(* Logix 5000 project; controller CarbonScout_MK6 vendor 1 type 14 code 154 rev 32.11; software revision 32.00; part 7 of 17 *)

        [2,16].Day := 20, [2,16].Month := 11, [2,16].Year := 2021, [2,16].Sample_DO := 5.8144927, [2,16].Sample_pH := 9.2394, [2,16].Sample_VOL := 17.577055, [2,16].Density := 412.98294, [2,16].EmptyDist := 1410.0, [2,16].FullDist := 1326.2568, [2,16].Carbon_mLperL := 12.587779, [2,16].Slurry_Weight := -10.52187, [2,16].Sample_Tank := 2, [2,16].Carbon_Height := 83.743164, [2,16].Sample_FlowRate := 1.5023123, [2,16].Sample_FillTime := 11.700001, [2,16].DisplacedCarbonVol := 1512.862, [2,16].DisplacedCarbonMass := 756.431, [2,16].SampleDuration := 964, [2,17].Run_ID := 2610, [2,17].Carbon_VOL_ml := 220.35596, [2,17].Carbon_MASS := 110.17798, [2,17].Carbon_DIST := 6.5356975, [2,17].Hour := 1, [2,17].Min := 21, [2,17].Day := 20, [2,17].Month := 11, [2,17].Year := 2021, [2,17].Sample_DO := 6.0987396, [2,17].Sample_pH := 9.333745, [2,17].Sample_VOL := 16.857876, [2,17].Density := 402.41284, [2,17].EmptyDist := 1410.0, [2,17].FullDist := 1326.5975, [2,17].Carbon_mLperL := 13.071395, [2,17].Slurry_Weight := -10.52187, [2,17].Sample_Tank := 2, [2,17].Carbon_Height := 83.402466, [2,17].Sample_FlowRate := 1.9698381, [2,17].Sample_FillTime := 8.558001, [2,17].DisplacedCarbonVol := 2059.8826, [2,17].DisplacedCarbonMass := 1029.9413, [2,17].SampleDuration := 1054, [2,18].Run_ID := 2601, [2,18].Carbon_VOL_ml := 180.58542, [2,18].Carbon_MASS := 90.29271, [2,18].Carbon_DIST := 5.3398423, [2,18].Hour := 23, [2,18].Min := 4, [2,18].Day := 19, [2,18].Month := 11, [2,18].Year := 2021, [2,18].Sample_DO := 6.4815454, [2,18].Sample_pH := 9.355976, [2,18].Sample_VOL := 16.909246, [2,18].Density := 403.16788, [2,18].EmptyDist := 1410.0, [2,18].FullDist := 1341.6503, [2,18].Carbon_mLperL := 10.679685, [2,18].Slurry_Weight := -10.52187, [2,18].Sample_Tank := 2,
        [2,18].Carbon_Height := 68.34973, [2,18].Sample_FlowRate := 2.087561, [2,18].Sample_FillTime := 8.100001, [2,18].DisplacedCarbonVol := 1783.5593, [2,18].DisplacedCarbonMass := 891.77966, [2,18].SampleDuration := 876, [2,19].Run_ID := 2593, [2,19].Carbon_VOL_ml := 185.95343, [2,19].Carbon_MASS := 92.976715, [2,19].Carbon_DIST := 5.4190025, [2,19].Hour := 21, [2,19].Min := 7, [2,19].Day := 19, [2,19].Month := 11, [2,19].Year := 2021, [2,19].Sample_DO := 6.719078, [2,19].Sample_pH := 9.30912, [2,19].Sample_VOL := 17.157534, [2,19].Density := 406.81705, [2,19].EmptyDist := 1410.0, [2,19].FullDist := 1339.6185, [2,19].Carbon_mLperL := 10.838005, [2,19].Slurry_Weight := -10.52187, [2,19].Sample_Tank := 2, [2,19].Carbon_Height := 70.38147, [2,19].Sample_FlowRate := 2.3369017, [2,19].Sample_FillTime := 7.342001, [2,19].DisplacedCarbonVol := 2026.1881, [2,19].DisplacedCarbonMass := 1013.09406, [2,19].SampleDuration := 876, [3,0].Run_ID := 2785, [3,0].Hour := 22, [3,0].Min := 56, [3,0].Day := 21, [3,0].Month := 11, [3,0].Year := 2021, [3,0].Sample_DO := 5.975054, [3,0].Sample_pH := 9.085041, [3,0].Sample_VOL := 17.71404, [3,0].Density := 414.99634, [3,0].EmptyDist := 1410.0, [3,0].FullDist := 1441.737, [3,0].ErrorFlag := 1, [3,0].Slurry_Weight := -10.52187, [3,0].Sample_Tank := 3, [3,0].Carbon_Height := -31.73706, [3,0].Sample_FlowRate := 1.3902087, [3,0].Sample_FillTime := 12.742001, [3,0].SampleDuration := 926, [3,1].Run_ID := 2784, [3,1].Carbon_VOL_ml := 131.5602, [3,1].Carbon_MASS := 65.7801, [3,1].Carbon_DIST := 3.8647463, [3,1].Hour := 22, [3,1].Min := 41, [3,1].Day := 21, [3,1].Month := 11, [3,1].Year := 2021, [3,1].Sample_DO := 6.334731, [3,1].Sample_pH := 9.09235,
        [3,1].Sample_VOL := 17.020548, [3,1].Density := 404.8037, [3,1].EmptyDist := 1410.0, [3,1].FullDist := 1360.2058, [3,1].Carbon_mLperL := 7.7294927, [3,1].Slurry_Weight := -10.52187, [3,1].Sample_Tank := 3, [3,1].Carbon_Height := 49.79419, [3,1].Sample_FlowRate := 1.350837, [3,1].Sample_FillTime := 12.600001, [3,1].DisplacedCarbonVol := 1044.1285, [3,1].DisplacedCarbonMass := 522.0643, [3,1].SampleDuration := 941, [3,2].Run_ID := 2771, [3,2].Hour := 19, [3,2].Min := 27, [3,2].Day := 21, [3,2].Month := 11, [3,2].Year := 2021, [3,2].Sample_DO := 6.247068, [3,2].Sample_pH := 9.097762, [3,2].Sample_VOL := 17.619864, [3,2].Density := 413.61212, [3,2].EmptyDist := 1410.0, [3,2].FullDist := 1446.4924, [3,2].ErrorFlag := 1, [3,2].Slurry_Weight := -10.52187, [3,2].Sample_Tank := 3, [3,2].Carbon_Height := -36.49243, [3,2].Sample_FlowRate := 1.4161599, [3,2].Sample_FillTime := 12.442001, [3,2].SampleDuration := 925, [3,3].Run_ID := 2770, [3,3].Hour := 19, [3,3].Min := 12, [3,3].Day := 21, [3,3].Month := 11, [3,3].Year := 2021, [3,3].Sample_DO := 5.9098787, [3,3].Sample_pH := 9.116793, [3,3].Sample_VOL := 16.515411, [3,3].Density := 397.3795, [3,3].EmptyDist := 1410.0, [3,3].FullDist := 1444.21, [3,3].Slurry_Weight := -10.52187, [3,3].Sample_Tank := 3, [3,3].Carbon_Height := -34.20996, [3,3].Sample_FlowRate := 1.428916, [3,3].Sample_FillTime := 11.558001, [3,3].SampleDuration := 988, [3,4].Run_ID := 2748, [3,4].Carbon_VOL_ml := 107.38028, [3,4].Carbon_MASS := 53.69014, [3,4].Carbon_DIST := 3.1075363, [3,4].Hour := 13, [3,4].Min := 17, [3,4].Day := 21, [3,4].Month := 11, [3,4].Year := 2021, [3,4].Sample_DO := 6.1838565,
        [3,4].Sample_pH := 9.131414, [3,4].Sample_VOL := 17.277397, [3,4].Density := 408.57877, [3,4].EmptyDist := 1410.0, [3,4].FullDist := 1369.3577, [3,4].ErrorFlag := 1, [3,4].Carbon_mLperL := 6.2150726, [3,4].Slurry_Weight := -10.52187, [3,4].Sample_Tank := 3, [3,4].Carbon_Height := 40.642334, [3,4].Sample_FlowRate := 1.1410247, [3,4].Sample_FillTime := 15.142001, [3,4].DisplacedCarbonVol := 709.15515, [3,4].DisplacedCarbonMass := 354.57758, [3,4].SampleDuration := 928, [3,5].Run_ID := 2747, [3,5].Carbon_VOL_ml := 89.66557, [3,5].Carbon_MASS := 44.832787, [3,5].Carbon_DIST := 2.55687, [3,5].Hour := 13, [3,5].Min := 1, [3,5].Day := 21, [3,5].Month := 11, [3,5].Year := 2021, [3,5].Sample_DO := 5.9852405, [3,5].Sample_pH := 9.164311, [3,5].Sample_VOL := 17.534246, [3,5].Density := 412.35376, [3,5].EmptyDist := 1410.0, [3,5].FullDist := 1376.0625, [3,5].Carbon_mLperL := 5.11374, [3,5].Slurry_Weight := -10.52187, [3,5].Sample_Tank := 3, [3,5].Carbon_Height := 33.9375, [3,5].Sample_FlowRate := 1.1354905, [3,5].Sample_FillTime := 15.442001, [3,5].DisplacedCarbonVol := 580.66034, [3,5].DisplacedCarbonMass := 290.33017, [3,5].SampleDuration := 876, [3,6].Run_ID := 2734, [3,6].Carbon_VOL_ml := 232.73778, [3,6].Carbon_MASS := 116.36889, [3,6].Carbon_DIST := 6.594802, [3,6].Hour := 9, [3,6].Min := 47, [3,6].Day := 21, [3,6].Month := 11, [3,6].Year := 2021, [3,6].Sample_DO := 5.8418803, [3,6].Sample_pH := 9.115876, [3,6].Sample_VOL := 17.645548, [3,6].Density := 413.98962, [3,6].EmptyDist := 1410.0, [3,6].FullDist := 1321.9111, [3,6].ErrorFlag := 1, [3,6].Carbon_mLperL := 13.189604, [3,6].Slurry_Weight := -10.52187, [3,6].Sample_Tank := 3, [3,6].Carbon_Height := 88.08887, [3,6].Sample_FlowRate := 1.2389796,
        [3,6].Sample_FillTime := 14.242001, [3,6].DisplacedCarbonVol := 1634.165, [3,6].DisplacedCarbonMass := 817.0825, [3,6].SampleDuration := 927, [3,7].Run_ID := 2733, [3,7].Carbon_VOL_ml := 232.98547, [3,7].Carbon_MASS := 116.49274, [3,7].Carbon_DIST := 6.776072, [3,7].Hour := 9, [3,7].Min := 31, [3,7].Day := 21, [3,7].Month := 11, [3,7].Year := 2021, [3,7].Sample_DO := 6.0491557, [3,7].Sample_pH := 9.1932335, [3,7].Sample_VOL := 17.19178, [3,7].Density := 407.3204, [3,7].EmptyDist := 1410.0, [3,7].FullDist := 1321.8174, [3,7].Carbon_mLperL := 13.552144, [3,7].Slurry_Weight := -10.52187, [3,7].Sample_Tank := 3, [3,7].Carbon_Height := 88.18262, [3,7].Sample_FlowRate := 1.3326961, [3,7].Sample_FillTime := 12.900001, [3,7].DisplacedCarbonVol := 1806.0889, [3,7].DisplacedCarbonMass := 903.04443, [3,7].SampleDuration := 877, [3,8].Run_ID := 2723, [3,8].Carbon_VOL_ml := 140.70815, [3,8].Carbon_MASS := 70.35407, [3,8].Carbon_DIST := 3.9870722, [3,8].Hour := 6, [3,8].Min := 9, [3,8].Day := 21, [3,8].Month := 11, [3,8].Year := 2021, [3,8].Sample_DO := 5.5555353, [3,8].Sample_pH := 9.267746, [3,8].Sample_VOL := 17.645548, [3,8].Density := 413.98962, [3,8].EmptyDist := 1410.0, [3,8].FullDist := 1356.7434, [3,8].Carbon_mLperL := 7.9741445, [3,8].Slurry_Weight := -10.52187, [3,8].Sample_Tank := 3, [3,8].Carbon_Height := 53.25659, [3,8].Sample_FlowRate := 1.5896888, [3,8].Sample_FillTime := 11.100001, [3,8].DisplacedCarbonVol := 1267.6407, [3,8].DisplacedCarbonMass := 633.8204, [3,8].SampleDuration := 872, [3,9].Run_ID := 2712, [3,9].Carbon_VOL_ml := 180.66768, [3,9].Carbon_MASS := 90.33384, [3,9].Carbon_DIST := 5.0995617, [3,9].Hour := 3, [3,9].Min := 23, [3,9].Day := 21, [3,9].Month := 11,
        [3,9].Year := 2021, [3,9].Sample_DO := 6.18531, [3,9].Sample_pH := 9.155949, [3,9].Sample_VOL := 17.71404, [3,9].Density := 414.99634, [3,9].EmptyDist := 1410.0, [3,9].FullDist := 1341.6191, [3,9].Carbon_mLperL := 10.199123, [3,9].Slurry_Weight := -10.52187, [3,9].Sample_Tank := 3, [3,9].Carbon_Height := 68.38086, [3,9].Sample_FlowRate := 1.4958655, [3,9].Sample_FillTime := 11.842001, [3,9].DisplacedCarbonVol := 1525.6516, [3,9].DisplacedCarbonMass := 762.8258, [3,9].SampleDuration := 874, [3,10].Run_ID := 2701, [3,10].Carbon_VOL_ml := 169.69102, [3,10].Carbon_MASS := 84.84551, [3,10].Carbon_DIST := 4.8721514, [3,10].Min := 44, [3,10].Day := 21, [3,10].Month := 11, [3,10].Year := 2021, [3,10].Sample_DO := 5.931424, [3,10].Sample_pH := 9.080997, [3,10].Sample_VOL := 17.414383, [3,10].Density := 410.59213, [3,10].EmptyDist := 1410.0, [3,10].FullDist := 1345.7737, [3,10].ErrorFlag := 1, [3,10].Carbon_mLperL := 9.744303, [3,10].Slurry_Weight := -10.52187, [3,10].Sample_Tank := 3, [3,10].Carbon_Height := 64.22632, [3,10].Sample_FlowRate := 1.3666915, [3,10].Sample_FillTime := 12.742001, [3,10].DisplacedCarbonVol := 1331.7456, [3,10].DisplacedCarbonMass := 665.8728, [3,10].SampleDuration := 927, [3,11].Run_ID := 2700, [3,11].Carbon_VOL_ml := 162.94458, [3,11].Carbon_MASS := 81.47229, [3,11].Carbon_DIST := 4.5357313, [3,11].Min := 28, [3,11].Day := 21, [3,11].Month := 11, [3,11].Year := 2021, [3,11].Sample_DO := 6.049618, [3,11].Sample_pH := 9.090882, [3,11].Sample_VOL := 17.962328, [3,11].Density := 418.64548, [3,11].EmptyDist := 1410.0, [3,11].FullDist := 1348.3271, [3,11].Carbon_mLperL := 9.071463, [3,11].Slurry_Weight := -10.52187, [3,11].Sample_Tank := 3, [3,11].Carbon_Height := 61.67285, [3,11].Sample_FlowRate := 1.3305427, [3,11].Sample_FillTime := 13.500001,
        [3,11].DisplacedCarbonVol := 1206.997, [3,11].DisplacedCarbonMass := 603.4985, [3,11].SampleDuration := 877, [3,12].Run_ID := 2688, [3,12].Carbon_VOL_ml := 2.5427434, [3,12].Carbon_MASS := 1.2713717, [3,12].Carbon_DIST := 0.071323834, [3,12].Hour := 21, [3,12].Min := 31, [3,12].Day := 20, [3,12].Month := 11, [3,12].Year := 2021, [3,12].Sample_DO := 5.966387, [3,12].Sample_pH := 9.127291, [3,12].Sample_VOL := 17.825342, [3,12].Density := 416.63214, [3,12].EmptyDist := 1410.0, [3,12].FullDist := 1409.0376, [3,12].ErrorFlag := 1, [3,12].Carbon_mLperL := 0.14264767, [3,12].Slurry_Weight := -10.52187, [3,12].Sample_Tank := 3, [3,12].Carbon_Height := 0.96240234, [3,12].Sample_FlowRate := 1.5052644, [3,12].Sample_FillTime := 11.842001, [3,12].DisplacedCarbonVol := 21.472246, [3,12].DisplacedCarbonMass := 10.736123, [3,12].SampleDuration := 926, [3,13].Run_ID := 2687, [3,13].Carbon_VOL_ml := 87.715294, [3,13].Carbon_MASS := 43.857647, [3,13].Carbon_DIST := 2.512297, [3,13].Hour := 21, [3,13].Min := 16, [3,13].Day := 20, [3,13].Month := 11, [3,13].Year := 2021, [3,13].Sample_DO := 6.0653386, [3,13].Sample_pH := 9.228728, [3,13].Sample_VOL := 17.457191, [3,13].Density := 411.22125, [3,13].EmptyDist := 1410.0, [3,13].FullDist := 1376.8007, [3,13].Carbon_mLperL := 5.024594, [3,13].Slurry_Weight := -10.52187, [3,13].Sample_Tank := 3, [3,13].Carbon_Height := 33.19934, [3,13].Sample_FlowRate := 1.4741758, [3,13].Sample_FillTime := 11.842001, [3,13].DisplacedCarbonVol := 740.7135, [3,13].DisplacedCarbonMass := 370.35675, [3,13].SampleDuration := 873, [3,14].Run_ID := 2676, [3,14].Carbon_VOL_ml := 316.40967, [3,14].Carbon_MASS := 158.20483, [3,14].Carbon_DIST := 9.120595, [3,14].Hour := 18, [3,14].Min := 27, [3,14].Day := 20, [3,14].Month := 11,
        [3,14].Year := 2021, [3,14].Sample_DO := 5.684902, [3,14].Sample_pH := 9.152988, [3,14].Sample_VOL := 17.34589, [3,14].Density := 409.58542, [3,14].EmptyDist := 1410.0, [3,14].FullDist := 1290.2422, [3,14].ErrorFlag := 1, [3,14].Carbon_mLperL := 18.24119, [3,14].Slurry_Weight := -10.52187, [3,14].Sample_Tank := 3, [3,14].Carbon_Height := 119.75781, [3,14].Sample_FlowRate := 1.5626926, [3,14].Sample_FillTime := 11.100001, [3,14].DisplacedCarbonVol := 2850.5374, [3,14].DisplacedCarbonMass := 1425.2687, [3,14].SampleDuration := 925, [3,15].Run_ID := 2675, [3,15].Carbon_VOL_ml := 318.91373, [3,15].Carbon_MASS := 159.45686, [3,15].Carbon_DIST := 9.321602, [3,15].Hour := 18, [3,15].Min := 11, [3,15].Day := 20, [3,15].Month := 11, [3,15].Year := 2021, [3,15].Sample_DO := 5.655153, [3,15].Sample_pH := 9.277301, [3,15].Sample_VOL := 17.106165, [3,15].Density := 406.06207, [3,15].EmptyDist := 1410.0, [3,15].FullDist := 1289.2944, [3,15].Carbon_mLperL := 18.643204, [3,15].Slurry_Weight := -10.52187, [3,15].Sample_Tank := 3, [3,15].Carbon_Height := 120.70557, [3,15].Sample_FlowRate := 1.5005407, [3,15].Sample_FillTime := 11.400001, [3,15].DisplacedCarbonVol := 2797.4888, [3,15].DisplacedCarbonMass := 1398.7444, [3,15].SampleDuration := 871, [3,16].Run_ID := 2663, [3,16].Carbon_VOL_ml := 193.90451, [3,16].Carbon_MASS := 96.952255, [3,16].Carbon_DIST := 5.6338425, [3,16].Hour := 15, [3,16].Min := 17, [3,16].Day := 20, [3,16].Month := 11, [3,16].Year := 2021, [3,16].Sample_DO := 5.4973636, [3,16].Sample_pH := 9.102047, [3,16].Sample_VOL := 17.208904, [3,16].Density := 407.57208, [3,16].EmptyDist := 1410.0, [3,16].FullDist := 1336.6091, [3,16].ErrorFlag := 1, [3,16].Carbon_mLperL := 11.267685, [3,16].Slurry_Weight := -10.52187, [3,16].Sample_Tank := 3,
        [3,16].Carbon_Height := 73.39087, [3,16].Sample_FlowRate := 1.4173038, [3,16].Sample_FillTime := 12.142001, [3,16].DisplacedCarbonVol := 1596.9734, [3,16].DisplacedCarbonMass := 798.4867, [3,16].SampleDuration := 925, [3,17].Run_ID := 2662, [3,17].Hour := 15, [3,17].Min := 1, [3,17].Day := 20, [3,17].Month := 11, [3,17].Year := 2021, [3,17].Sample_DO := 5.5800033, [3,17].Sample_pH := 9.173197, [3,17].Sample_VOL := 17.55993, [3,17].Density := 412.73126, [3,17].EmptyDist := 1410.0, [3,17].FullDist := 1430.6094, [3,17].Slurry_Weight := -10.52187, [3,17].Sample_Tank := 3, [3,17].Carbon_Height := -20.609375, [3,17].Sample_FlowRate := 1.4276365, [3,17].Sample_FillTime := 12.300001, [3,17].SampleDuration := 872, [3,18].Run_ID := 2650, [3,18].Carbon_VOL_ml := 169.7033, [3,18].Carbon_MASS := 84.85165, [3,18].Carbon_DIST := 5.056465, [3,18].Hour := 12, [3,18].Day := 20, [3,18].Month := 11, [3,18].Year := 2021, [3,18].Sample_DO := 5.6071215, [3,18].Sample_pH := 9.084224, [3,18].Sample_VOL := 16.780823, [3,18].Density := 401.2804, [3,18].EmptyDist := 1410.0, [3,18].FullDist := 1345.769, [3,18].Carbon_mLperL := 10.11293, [3,18].Slurry_Weight := -10.52187, [3,18].Sample_Tank := 3, [3,18].Carbon_Height := 64.23096, [3,18].Sample_FlowRate := 1.1187215, [3,18].Sample_FillTime := 15.000001, [3,18].DisplacedCarbonVol := 1131.3552, [3,18].DisplacedCarbonMass := 565.6776, [3,18].SampleDuration := 878, [3,19].Run_ID := 2640, [3,19].Carbon_VOL_ml := 185.8657, [3,19].Carbon_MASS := 92.93285, [3,19].Carbon_DIST := 5.354986, [3,19].Hour := 9, [3,19].Min := 28, [3,19].Day := 20, [3,19].Month := 11, [3,19].Year := 2021, [3,19].Sample_DO := 6.2630897, [3,19].Sample_pH := 9.137375, [3,19].Sample_VOL := 17.354452, [3,19].Density := 409.71127,
        [3,19].EmptyDist := 1410.0, [3,19].FullDist := 1339.6517, [3,19].Carbon_mLperL := 10.709972, [3,19].Slurry_Weight := -10.52187, [3,19].Sample_Tank := 3, [3,19].Carbon_Height := 70.34827, [3,19].Sample_FlowRate := 1.1226841, [3,19].Sample_FillTime := 15.458001, [3,19].DisplacedCarbonVol := 1202.3916, [3,19].DisplacedCarbonMass := 601.1958, [3,19].SampleDuration := 879, [4,0].Run_ID := 2787, [4,0].Hour := 23, [4,0].Min := 27, [4,0].Day := 21, [4,0].Month := 11, [4,0].Year := 2021, [4,0].Sample_DO := 5.6127687, [4,0].Sample_pH := 9.112585, [4,0].Sample_VOL := 17.34589, [4,0].Density := 409.58542, [4,0].EmptyDist := 1410.0, [4,0].FullDist := 1447.225, [4,0].ErrorFlag := 1, [4,0].Slurry_Weight := -10.52187, [4,0].Sample_Tank := 4, [4,0].Carbon_Height := -37.224976, [4,0].Sample_FlowRate := 1.464777, [4,0].Sample_FillTime := 11.842001, [4,0].SampleDuration := 926, [4,1].Run_ID := 2786, [4,1].Hour := 23, [4,1].Min := 11, [4,1].Day := 21, [4,1].Month := 11, [4,1].Year := 2021, [4,1].Sample_DO := 5.879518, [4,1].Sample_pH := 9.193804, [4,1].Sample_VOL := 17.208904, [4,1].Density := 407.57208, [4,1].EmptyDist := 1410.0, [4,1].FullDist := 1447.1635, [4,1].Slurry_Weight := -10.52187, [4,1].Sample_Tank := 4, [4,1].Carbon_Height := -37.163452, [4,1].Sample_FlowRate := 1.4340752, [4,1].Sample_FillTime := 12.000001, [4,1].SampleDuration := 927, [4,2].Run_ID := 2773, [4,2].Hour := 19, [4,2].Min := 58, [4,2].Day := 21, [4,2].Month := 11, [4,2].Year := 2021, [4,2].Sample_DO := 5.849701, [4,2].Sample_pH := 9.101484, [4,2].Sample_VOL := 17.722603, [4,2].Density := 415.12213, [4,2].EmptyDist := 1410.0, [4,2].FullDist := 1447.1489,
        [4,2].ErrorFlag := 1, [4,2].Slurry_Weight := -10.52187, [4,2].Sample_Tank := 4, [4,2].Carbon_Height := -37.148926, [4,2].Sample_FlowRate := 1.3127853, [4,2].Sample_FillTime := 13.500001, [4,2].SampleDuration := 927, [4,3].Run_ID := 2772, [4,3].Hour := 19, [4,3].Min := 43, [4,3].Day := 21, [4,3].Month := 11, [4,3].Year := 2021, [4,3].Sample_DO := 5.853695, [4,3].Sample_pH := 9.12075, [4,3].Sample_VOL := 17.465754, [4,3].Density := 411.34714, [4,3].EmptyDist := 1410.0, [4,3].FullDist := 1440.5786, [4,3].Slurry_Weight := -10.52187, [4,3].Sample_Tank := 4, [4,3].Carbon_Height := -30.578613, [4,3].Sample_FlowRate := 1.3391927, [4,3].Sample_FillTime := 13.042001, [4,3].SampleDuration := 926, [4,4].Run_ID := 2750, [4,4].Carbon_VOL_ml := 178.94606, [4,4].Carbon_MASS := 89.47303, [4,4].Carbon_DIST := 5.1940603, [4,4].Hour := 13, [4,4].Min := 48, [4,4].Day := 21, [4,4].Month := 11, [4,4].Year := 2021, [4,4].Sample_DO := 5.656315, [4,4].Sample_pH := 9.1106205, [4,4].Sample_VOL := 17.226028, [4,4].Density := 407.82376, [4,4].EmptyDist := 1410.0, [4,4].FullDist := 1342.2708, [4,4].ErrorFlag := 1, [4,4].Carbon_mLperL := 10.388121, [4,4].Slurry_Weight := -10.52187, [4,4].Sample_Tank := 4, [4,4].Carbon_Height := 67.72925, [4,4].Sample_FlowRate := 1.0350935, [4,4].Sample_FillTime := 16.642002, [4,4].DisplacedCarbonVol := 1075.2677, [4,4].DisplacedCarbonMass := 537.63385, [4,4].SampleDuration := 931, [4,5].Run_ID := 2749, [4,5].Hour := 13, [4,5].Min := 32, [4,5].Day := 21, [4,5].Month := 11, [4,5].Year := 2021, [4,5].Sample_DO := 5.5927024, [4,5].Sample_pH := 9.106966, [4,5].Sample_VOL := 17.226028, [4,5].Density := 407.82376,
        [4,5].EmptyDist := 1410.0, [4,5].FullDist := 1415.5074, [4,5].Slurry_Weight := -10.52187, [4,5].Sample_Tank := 4, [4,5].Carbon_Height := -5.5074463, [4,5].Sample_FlowRate := 1.083398, [4,5].Sample_FillTime := 15.900001, [4,5].SampleDuration := 928, [4,6].Run_ID := 2736, [4,6].Carbon_VOL_ml := 185.82217, [4,6].Carbon_MASS := 92.91109, [4,6].Carbon_DIST := 5.270527, [4,6].Hour := 10, [4,6].Min := 17, [4,6].Day := 21, [4,6].Month := 11, [4,6].Year := 2021, [4,6].Sample_DO := 5.6108036, [4,6].Sample_pH := 9.108102, [4,6].Sample_VOL := 17.628426, [4,6].Density := 413.73798, [4,6].EmptyDist := 1410.0, [4,6].FullDist := 1339.6682, [4,6].ErrorFlag := 1, [4,6].Carbon_mLperL := 10.541054, [4,6].Slurry_Weight := -10.52187, [4,6].Sample_Tank := 4, [4,6].Carbon_Height := 70.33179, [4,6].Sample_FlowRate := 1.3516657, [4,6].Sample_FillTime := 13.042001, [4,6].DisplacedCarbonVol := 1424.7982, [4,6].DisplacedCarbonMass := 712.3991, [4,6].SampleDuration := 928, [4,7].Run_ID := 2735, [4,7].Carbon_VOL_ml := 104.513084, [4,7].Carbon_MASS := 52.256542, [4,7].Carbon_DIST := 2.9301796, [4,7].Hour := 10, [4,7].Min := 2, [4,7].Day := 21, [4,7].Month := 11, [4,7].Year := 2021, [4,7].Sample_DO := 5.9035196, [4,7].Sample_pH := 9.203241, [4,7].Sample_VOL := 17.833904, [4,7].Density := 416.75797, [4,7].EmptyDist := 1410.0, [4,7].FullDist := 1370.4429, [4,7].Carbon_mLperL := 5.860359, [4,7].Slurry_Weight := -10.52187, [4,7].Sample_Tank := 4, [4,7].Carbon_Height := 39.55713, [4,7].Sample_FlowRate := 1.3210299, [4,7].Sample_FillTime := 13.500001, [4,7].DisplacedCarbonVol := 774.171, [4,7].DisplacedCarbonMass := 387.0855, [4,7].SampleDuration := 928, [4,8].Run_ID := 2725, [4,8].Carbon_VOL_ml := 289.29868, [4,8].Carbon_MASS := 144.64934,
        [4,8].Carbon_DIST := 8.66857, [4,8].Hour := 6, [4,8].Min := 49, [4,8].Day := 21, [4,8].Month := 11, [4,8].Year := 2021, [4,8].Sample_DO := 5.661371, [4,8].Sample_pH := 9.14287, [4,8].Sample_VOL := 16.686644, [4,8].Density := 399.89615, [4,8].EmptyDist := 1410.0, [4,8].FullDist := 1300.5034, [4,8].ErrorFlag := 1, [4,8].Carbon_mLperL := 17.33714, [4,8].Slurry_Weight := -10.52187, [4,8].Sample_Tank := 4, [4,8].Carbon_Height := 109.49658, [4,8].Sample_FlowRate := 1.4637406, [4,8].Sample_FillTime := 11.400001, [4,8].DisplacedCarbonVol := 2537.7075, [4,8].DisplacedCarbonMass := 1268.8538, [4,8].SampleDuration := 926, [4,9].Run_ID := 2724, [4,9].Carbon_VOL_ml := 287.28967, [4,9].Carbon_MASS := 143.64484, [4,9].Carbon_DIST := 8.1169405, [4,9].Hour := 6, [4,9].Min := 24, [4,9].Day := 21, [4,9].Month := 11, [4,9].Year := 2021, [4,9].Sample_DO := 5.696142, [4,9].Sample_pH := 9.273345, [4,9].Sample_VOL := 17.696918, [4,9].Density := 414.74466, [4,9].EmptyDist := 1410.0, [4,9].FullDist := 1301.2638, [4,9].Carbon_mLperL := 16.233881, [4,9].Slurry_Weight := -10.52187, [4,9].Sample_Tank := 4, [4,9].Carbon_Height := 108.736206, [4,9].Sample_FlowRate := 1.4924033, [4,9].Sample_FillTime := 11.858001, [4,9].DisplacedCarbonVol := 2422.75, [4,9].DisplacedCarbonMass := 1211.375, [4,9].SampleDuration := 924, [4,10].Run_ID := 2714, [4,10].Hour := 3, [4,10].Min := 58, [4,10].Day := 21, [4,10].Month := 11, [4,10].Year := 2021, [4,10].Sample_DO := 5.938393, [4,10].Sample_pH := 9.215282, [4,10].Sample_VOL := 6.308176, [4,10].Density := 247.35901, [4,10].EmptyDist := 1410.0, [4,10].FullDist := 1412.2761, [4,10].ErrorFlag := 1, [4,10].Slurry_Weight := -10.52187,
        [4,10].Sample_Tank := 4, [4,10].Carbon_Height := -2.276123, [4,10].Sample_FlowRate := 0.042054508, [4,10].Sample_FillTime := 150.0, [4,10].SampleDuration := 1063, [4,11].Run_ID := 2713, [4,11].Hour := 3, [4,11].Min := 41, [4,11].Day := 21, [4,11].Month := 11, [4,11].Year := 2021, [4,11].Sample_DO := 5.407501, [4,11].Sample_pH := 9.241049, [4,11].Sample_VOL := 9.872117, [4,11].Density := 299.7399, [4,11].EmptyDist := 1410.0, [4,11].FullDist := 1412.6694, [4,11].Slurry_Weight := -10.52187, [4,11].Sample_Tank := 4, [4,11].Carbon_Height := -2.6694336, [4,11].Sample_FlowRate := 0.065814115, [4,11].Sample_FillTime := 150.0, [4,11].SampleDuration := 925, [4,12].Run_ID := 2703, [4,12].Carbon_VOL_ml := 268.5752, [4,12].Carbon_MASS := 134.2876, [4,12].Carbon_DIST := 7.7455764, [4,12].Hour := 1, [4,12].Min := 15, [4,12].Day := 21, [4,12].Month := 11, [4,12].Year := 2021, [4,12].Sample_DO := 5.7639284, [4,12].Sample_pH := 9.075916, [4,12].Sample_VOL := 17.337328, [4,12].Density := 409.45953, [4,12].EmptyDist := 1410.0, [4,12].FullDist := 1308.347, [4,12].ErrorFlag := 1, [4,12].Carbon_mLperL := 15.491153, [4,12].Slurry_Weight := -10.52187, [4,12].Sample_Tank := 4, [4,12].Carbon_Height := 101.652954, [4,12].Sample_FlowRate := 1.1227384, [4,12].Sample_FillTime := 15.442001, [4,12].DisplacedCarbonVol := 1739.2512, [4,12].DisplacedCarbonMass := 869.6256, [4,12].SampleDuration := 928, [4,13].Run_ID := 2702, [4,13].Carbon_VOL_ml := 227.51007, [4,13].Carbon_MASS := 113.755035, [4,13].Carbon_DIST := 6.8558245, [4,13].Min := 59, [4,13].Day := 21, [4,13].Month := 11, [4,13].Year := 2021, [4,13].Sample_DO := 5.537921, [4,13].Sample_pH := 9.081407, [4,13].Sample_VOL := 16.592466, [4,13].Density := 398.512,
        [4,13].EmptyDist := 1410.0, [4,13].FullDist := 1323.8898, [4,13].Carbon_mLperL := 13.711649, [4,13].Slurry_Weight := -10.52187, [4,13].Sample_Tank := 4, [4,13].Carbon_Height := 86.11023, [4,13].Sample_FlowRate := 1.2023525, [4,13].Sample_FillTime := 13.800001, [4,13].DisplacedCarbonVol := 1648.6235, [4,13].DisplacedCarbonMass := 824.31177, [4,13].SampleDuration := 926, [4,14].Run_ID := 2690, [4,14].Hour := 22, [4,14].Min := 2, [4,14].Day := 20, [4,14].Month := 11, [4,14].Year := 2021, [4,14].Sample_DO := 5.56772, [4,14].Sample_pH := 9.115578, [4,14].Sample_VOL := 18.005136, [4,14].Density := 419.27466, [4,14].EmptyDist := 1410.0, [4,14].FullDist := 1443.7524, [4,14].ErrorFlag := 1, [4,14].Slurry_Weight := -10.52187, [4,14].Sample_Tank := 4, [4,14].Carbon_Height := -33.75244, [4,14].Sample_FlowRate := 1.4638321, [4,14].Sample_FillTime := 12.300001, [4,14].SampleDuration := 926, [4,15].Run_ID := 2689, [4,15].Hour := 21, [4,15].Min := 47, [4,15].Day := 20, [4,15].Month := 11, [4,15].Year := 2021, [4,15].Sample_DO := 5.91934, [4,15].Sample_pH := 9.220631, [4,15].Sample_VOL := 17.671232, [4,15].Density := 414.36716, [4,15].EmptyDist := 1410.0, [4,15].FullDist := 1427.2971, [4,15].Slurry_Weight := -10.52187, [4,15].Sample_Tank := 4, [4,15].Carbon_Height := -17.29712, [4,15].Sample_FlowRate := 1.3868492, [4,15].Sample_FillTime := 12.742001, [4,15].SampleDuration := 925, [4,16].Run_ID := 2678, [4,16].Carbon_VOL_ml := 98.888336, [4,16].Carbon_MASS := 49.444168, [4,16].Carbon_DIST := 2.8889837, [4,16].Hour := 18, [4,16].Min := 57, [4,16].Day := 20, [4,16].Month := 11, [4,16].Year := 2021, [4,16].Sample_DO := 5.5482745, [4,16].Sample_pH := 9.139303, [4,16].Sample_VOL := 17.114727,
        [4,16].Density := 406.18787, [4,16].EmptyDist := 1410.0, [4,16].FullDist := 1372.5718, [4,16].ErrorFlag := 1, [4,16].Carbon_mLperL := 5.7779675, [4,16].Slurry_Weight := -10.52187, [4,16].Sample_Tank := 4, [4,16].Carbon_Height := 37.428223, [4,16].Sample_FlowRate := 1.4452564, [4,16].Sample_FillTime := 11.842001, [4,16].DisplacedCarbonVol := 835.0644, [4,16].DisplacedCarbonMass := 417.5322, [4,16].SampleDuration := 927, [4,17].Run_ID := 2677, [4,17].Carbon_VOL_ml := 100.89216, [4,17].Carbon_MASS := 50.44608, [4,17].Carbon_DIST := 2.931394, [4,17].Hour := 18, [4,17].Min := 42, [4,17].Day := 20, [4,17].Month := 11, [4,17].Year := 2021, [4,17].Sample_DO := 5.484293, [4,17].Sample_pH := 9.246172, [4,17].Sample_VOL := 17.208904, [4,17].Density := 407.57208, [4,17].EmptyDist := 1410.0, [4,17].FullDist := 1371.8134, [4,17].Carbon_mLperL := 5.862788, [4,17].Slurry_Weight := -10.52187, [4,17].Sample_Tank := 4, [4,17].Carbon_Height := 38.186646, [4,17].Sample_FlowRate := 1.3990978, [4,17].Sample_FillTime := 12.300001, [4,17].DisplacedCarbonVol := 820.26135, [4,17].DisplacedCarbonMass := 410.13068, [4,17].SampleDuration := 923, [4,18].Run_ID := 2664, [4,18].Carbon_VOL_ml := 235.55049, [4,18].Carbon_MASS := 117.775246, [4,18].Carbon_DIST := 6.6422734, [4,18].Hour := 15, [4,18].Min := 32, [4,18].Day := 20, [4,18].Month := 11, [4,18].Year := 2021, [4,18].Sample_DO := 5.796437, [4,18].Sample_pH := 9.196914, [4,18].Sample_VOL := 17.731165, [4,18].Density := 415.24802, [4,18].EmptyDist := 1410.0, [4,18].FullDist := 1320.8466, [4,18].Carbon_mLperL := 13.284547, [4,18].Slurry_Weight := -10.52187, [4,18].Sample_Tank := 4, [4,18].Carbon_Height := 89.15344, [4,18].Sample_FlowRate := 1.3134196, [4,18].Sample_FillTime := 13.500001, [4,18].DisplacedCarbonVol := 1744.8185, [4,18].DisplacedCarbonMass := 872.40924,
        [4,18].SampleDuration := 925, [4,19].Run_ID := 2651, [4,19].Carbon_VOL_ml := 222.49846, [4,19].Carbon_MASS := 111.24923, [4,19].Carbon_DIST := 6.471071, [4,19].Hour := 12, [4,19].Min := 16, [4,19].Day := 20, [4,19].Month := 11, [4,19].Year := 2021, [4,19].Sample_DO := 5.488589, [4,19].Sample_pH := 9.0820465, [4,19].Sample_VOL := 17.19178, [4,19].Density := 407.3204, [4,19].EmptyDist := 1410.0, [4,19].FullDist := 1325.7866, [4,19].Carbon_mLperL := 12.942142, [4,19].Slurry_Weight := -10.52187, [4,19].Sample_Tank := 4, [4,19].Carbon_Height := 84.21338, [4,19].Sample_FlowRate := 1.3181858, [4,19].Sample_FillTime := 13.042001, [4,19].DisplacedCarbonVol := 1706.0148, [4,19].DisplacedCarbonMass := 853.0074, [4,19].SampleDuration := 933, [5,0].Run_ID := 2789, [5,0].Carbon_VOL_ml := 64.33941, [5,0].Carbon_MASS := 32.169704, [5,0].Carbon_DIST := 1.8038509, [5,0].Hour := 23, [5,0].Min := 51, [5,0].Day := 21, [5,0].Month := 11, [5,0].Year := 2021, [5,0].Sample_DO := 5.7689, [5,0].Sample_pH := 9.094793, [5,0].Sample_VOL := 17.833904, [5,0].Density := 416.75797, [5,0].EmptyDist := 1410.0, [5,0].FullDist := 1385.6482, [5,0].ErrorFlag := 1, [5,0].Carbon_mLperL := 3.6077018, [5,0].Slurry_Weight := -10.52187, [5,0].Sample_Tank := 5, [5,0].Carbon_Height := 24.351807, [5,0].Sample_FlowRate := 1.3210299, [5,0].Sample_FillTime := 13.500001, [5,0].DisplacedCarbonVol := 476.58823, [5,0].DisplacedCarbonMass := 238.29411, [5,0].SampleDuration := 736, [5,1].Run_ID := 2788, [5,1].Hour := 23, [5,1].Min := 39, [5,1].Day := 21, [5,1].Month := 11, [5,1].Year := 2021, [5,1].Sample_DO := 5.5441365, [5,1].Sample_pH := 9.097831, [5,1].Sample_VOL := 17.568493, [5,1].Density := 412.85712,
        [5,1].EmptyDist := 1410.0, [5,1].FullDist := 1447.2249, [5,1].Slurry_Weight := -10.52187, [5,1].Sample_Tank := 5, [5,1].Carbon_Height := -37.224854, [5,1].Sample_FlowRate := 1.3309463, [5,1].Sample_FillTime := 13.200001, [5,1].SampleDuration := 929, [5,2].Run_ID := 2775, [5,2].Hour := 20, [5,2].Min := 22, [5,2].Day := 21, [5,2].Month := 11, [5,2].Year := 2021, [5,2].Sample_DO := 6.10914, [5,2].Sample_pH := 9.091206, [5,2].Sample_VOL := 17.619864, [5,2].Density := 413.61212, [5,2].EmptyDist := 1410.0, [5,2].FullDist := 1446.9946, [5,2].ErrorFlag := 1, [5,2].Slurry_Weight := -10.52187, [5,2].Sample_Tank := 5, [5,2].Carbon_Height := -36.99463, [5,2].Sample_FlowRate := 1.2637973, [5,2].Sample_FillTime := 13.942001, [5,2].SampleDuration := 709, [5,3].Run_ID := 2774, [5,3].Hour := 20, [5,3].Min := 10, [5,3].Day := 21, [5,3].Month := 11, [5,3].Year := 2021, [5,3].Sample_DO := 5.794888, [5,3].Sample_pH := 9.094314, [5,3].Sample_VOL := 18.005136, [5,3].Density := 419.27466, [5,3].EmptyDist := 1410.0, [5,3].FullDist := 1441.797, [5,3].Slurry_Weight := -10.52187, [5,3].Sample_Tank := 5, [5,3].Carbon_Height := -31.796997, [5,3].Sample_FlowRate := 1.2914313, [5,3].Sample_FillTime := 13.942001, [5,3].SampleDuration := 928, [5,4].Run_ID := 2752, [5,4].Carbon_VOL_ml := 135.78748, [5,4].Carbon_MASS := 67.89374, [5,4].Carbon_DIST := 3.8476412, [5,4].Hour := 14, [5,4].Min := 11, [5,4].Day := 21, [5,4].Month := 11, [5,4].Year := 2021, [5,4].Sample_DO := 5.7564034, [5,4].Sample_pH := 9.065218, [5,4].Sample_VOL := 17.645548, [5,4].Density := 413.98962, [5,4].EmptyDist := 1410.0, [5,4].FullDist := 1358.6058,
        [5,4].ErrorFlag := 1, [5,4].Carbon_mLperL := 7.6952825, [5,4].Slurry_Weight := -10.52187, [5,4].Sample_Tank := 5, [5,4].Carbon_Height := 51.394165, [5,4].Sample_FlowRate := 1.2003773, [5,4].Sample_FillTime := 14.700001, [5,4].DisplacedCarbonVol := 923.7243, [5,4].DisplacedCarbonMass := 461.86215, [5,4].SampleDuration := 709, [5,5].Run_ID := 2751, [5,5].Carbon_VOL_ml := 56.890175, [5,5].Carbon_MASS := 28.445087, [5,5].Carbon_DIST := 1.597301, [5,5].Hour := 13, [5,5].Min := 59, [5,5].Day := 21, [5,5].Month := 11, [5,5].Year := 2021, [5,5].Sample_DO := 5.41634, [5,5].Sample_pH := 9.075092, [5,5].Sample_VOL := 17.80822, [5,5].Density := 416.3805, [5,5].EmptyDist := 1410.0, [5,5].FullDist := 1388.4677, [5,5].Carbon_mLperL := 3.194602, [5,5].Slurry_Weight := -10.52187, [5,5].Sample_Tank := 5, [5,5].Carbon_Height := 21.532349, [5,5].Sample_FlowRate := 1.2758431, [5,5].Sample_FillTime := 13.958001, [5,5].DisplacedCarbonVol := 407.58112, [5,5].DisplacedCarbonMass := 203.79056, [5,5].SampleDuration := 931, [5,6].Run_ID := 2737, [5,6].Carbon_VOL_ml := 135.99002, [5,6].Carbon_MASS := 67.99501, [5,6].Carbon_DIST := 3.9277039, [5,6].Hour := 10, [5,6].Min := 29, [5,6].Day := 21, [5,6].Month := 11, [5,6].Year := 2021, [5,6].Sample_DO := 5.6184325, [5,6].Sample_pH := 9.084645, [5,6].Sample_VOL := 17.311644, [5,6].Density := 409.0821, [5,6].EmptyDist := 1410.0, [5,6].FullDist := 1358.5292, [5,6].Carbon_mLperL := 7.8554077, [5,6].Slurry_Weight := -10.52187, [5,6].Sample_Tank := 5, [5,6].Carbon_Height := 51.470825, [5,6].Sample_FlowRate := 1.32575, [5,6].Sample_FillTime := 13.058001, [5,6].DisplacedCarbonVol := 1041.4307, [5,6].DisplacedCarbonMass := 520.71533, [5,6].SampleDuration := 927, [5,7].Run_ID := 2726, [5,7].Carbon_VOL_ml := 215.70909,
        [5,7].Carbon_MASS := 107.854546, [5,7].Carbon_DIST := 6.103397, [5,7].Hour := 7, [5,7].Min := 1, [5,7].Day := 21, [5,7].Month := 11, [5,7].Year := 2021, [5,7].Sample_DO := 5.6028533, [5,7].Sample_pH := 9.128891, [5,7].Sample_VOL := 17.671232, [5,7].Density := 414.36716, [5,7].EmptyDist := 1410.0, [5,7].FullDist := 1328.3563, [5,7].Carbon_mLperL := 12.206794, [5,7].Slurry_Weight := -10.52187, [5,7].Sample_Tank := 5, [5,7].Carbon_Height := 81.64368, [5,7].Sample_FlowRate := 1.4024786, [5,7].Sample_FillTime := 12.600001, [5,7].DisplacedCarbonVol := 1711.9766, [5,7].DisplacedCarbonMass := 855.9883, [5,7].SampleDuration := 917, [5,8].Run_ID := 2716, [5,8].Carbon_VOL_ml := 261.69327, [5,8].Carbon_MASS := 130.84663, [5,8].Carbon_DIST := 7.3510756, [5,8].Hour := 4, [5,8].Min := 22, [5,8].Day := 21, [5,8].Month := 11, [5,8].Year := 2021, [5,8].Sample_DO := 5.459996, [5,8].Sample_pH := 9.136606, [5,8].Sample_VOL := 17.799658, [5,8].Density := 416.2546, [5,8].EmptyDist := 1410.0, [5,8].FullDist := 1310.9518, [5,8].ErrorFlag := 1, [5,8].Carbon_mLperL := 14.702151, [5,8].Slurry_Weight := -10.52187, [5,8].Sample_Tank := 5, [5,8].Carbon_Height := 99.04822, [5,8].Sample_FlowRate := 1.3969281, [5,8].Sample_FillTime := 12.742001, [5,8].DisplacedCarbonVol := 2053.785, [5,8].DisplacedCarbonMass := 1026.8925, [5,8].SampleDuration := 707, [5,9].Run_ID := 2715, [5,9].Carbon_VOL_ml := 246.50035, [5,9].Carbon_MASS := 123.250175, [5,9].Carbon_DIST := 7.1762815, [5,9].Hour := 4, [5,9].Min := 10, [5,9].Day := 21, [5,9].Month := 11, [5,9].Year := 2021, [5,9].Sample_DO := 6.210182, [5,9].Sample_pH := 9.22908, [5,9].Sample_VOL := 17.174658, [5,9].Density := 407.0688,
        [5,9].EmptyDist := 1410.0, [5,9].FullDist := 1316.7021, [5,9].Carbon_mLperL := 14.352563, [5,9].Slurry_Weight := -10.52187, [5,9].Sample_Tank := 5, [5,9].Carbon_Height := 93.29785, [5,9].Sample_FlowRate := 1.3478776, [5,9].Sample_FillTime := 12.742001, [5,9].DisplacedCarbonVol := 1934.5499, [5,9].DisplacedCarbonMass := 967.27496, [5,9].SampleDuration := 1060, [5,10].Run_ID := 2704, [5,10].Carbon_VOL_ml := 142.71616, [5,10].Carbon_MASS := 71.35808, [5,10].Carbon_DIST := 4.0478983, [5,10].Hour := 1, [5,10].Min := 27, [5,10].Day := 21, [5,10].Month := 11, [5,10].Year := 2021, [5,10].Sample_DO := 5.615845, [5,10].Sample_pH := 9.072593, [5,10].Sample_VOL := 17.628426, [5,10].Density := 413.73798, [5,10].EmptyDist := 1410.0, [5,10].FullDist := 1355.9834, [5,10].Carbon_mLperL := 8.095797, [5,10].Slurry_Weight := -10.52187, [5,10].Sample_Tank := 5, [5,10].Carbon_Height := 54.0166, [5,10].Sample_FlowRate := 1.2644114, [5,10].Sample_FillTime := 13.942001, [5,10].DisplacedCarbonVol := 1023.64185, [5,10].DisplacedCarbonMass := 511.82092, [5,10].SampleDuration := 930, [5,11].Run_ID := 2692, [5,11].Carbon_VOL_ml := 122.65803, [5,11].Carbon_MASS := 61.329014, [5,11].Carbon_DIST := 3.5691223, [5,11].Hour := 22, [5,11].Min := 26, [5,11].Day := 20, [5,11].Month := 11, [5,11].Year := 2021, [5,11].Sample_DO := 5.5048094, [5,11].Sample_pH := 9.077998, [5,11].Sample_VOL := 17.18322, [5,11].Density := 407.1946, [5,11].EmptyDist := 1410.0, [5,11].FullDist := 1363.5752, [5,11].ErrorFlag := 1, [5,11].Carbon_mLperL := 7.1382446, [5,11].Slurry_Weight := -10.52187, [5,11].Sample_Tank := 5, [5,11].Carbon_Height := 46.424805, [5,11].Sample_FlowRate := 1.3637475, [5,11].Sample_FillTime := 12.600001, [5,11].DisplacedCarbonVol := 973.47626, [5,11].DisplacedCarbonMass := 486.73813, [5,11].SampleDuration := 709,
        [5,12].Run_ID := 2691, [5,12].Hour := 22, [5,12].Min := 14, [5,12].Day := 20, [5,12].Month := 11, [5,12].Year := 2021, [5,12].Sample_DO := 5.533932, [5,12].Sample_pH := 9.100771, [5,12].Sample_VOL := 17.773972, [5,12].Density := 415.87714, [5,12].EmptyDist := 1410.0, [5,12].FullDist := 1447.1218, [5,12].Slurry_Weight := -10.52187, [5,12].Sample_Tank := 5, [5,12].Carbon_Height := -37.121826, [5,12].Sample_FlowRate := 1.3165904, [5,12].Sample_FillTime := 13.500001, [5,12].SampleDuration := 926, [5,13].Run_ID := 2679, [5,13].Carbon_VOL_ml := 239.17108, [5,13].Carbon_MASS := 119.58554, [5,13].Carbon_DIST := 6.780384, [5,13].Hour := 19, [5,13].Min := 9, [5,13].Day := 20, [5,13].Month := 11, [5,13].Year := 2021, [5,13].Sample_DO := 5.8248835, [5,13].Sample_pH := 9.138246, [5,13].Sample_VOL := 17.636986, [5,13].Density := 413.8638, [5,13].EmptyDist := 1410.0, [5,13].FullDist := 1319.4762, [5,13].Carbon_mLperL := 13.560768, [5,13].Slurry_Weight := -10.52187, [5,13].Sample_Tank := 5, [5,13].Carbon_Height := 90.5238, [5,13].Sample_FlowRate := 1.3506651, [5,13].Sample_FillTime := 13.058001, [5,13].DisplacedCarbonVol := 1831.6057, [5,13].DisplacedCarbonMass := 915.80286, [5,13].SampleDuration := 926, [5,14].Run_ID := 2665, [5,14].Carbon_VOL_ml := 163.72314, [5,14].Carbon_MASS := 81.86157, [5,14].Carbon_DIST := 4.544407, [5,14].Hour := 15, [5,14].Min := 44, [5,14].Day := 20, [5,14].Month := 11, [5,14].Year := 2021, [5,14].Sample_DO := 5.5120296, [5,14].Sample_pH := 9.11399, [5,14].Sample_VOL := 18.013699, [5,14].Density := 419.40054, [5,14].EmptyDist := 1410.0, [5,14].FullDist := 1348.0325, [5,14].Carbon_mLperL := 9.088814, [5,14].Slurry_Weight := -10.52187, [5,14].Sample_Tank := 5,
        [5,14].Carbon_Height := 61.96753, [5,14].Sample_FlowRate := 1.2920454, [5,14].Sample_FillTime := 13.942001, [5,14].DisplacedCarbonVol := 1174.316, [5,14].DisplacedCarbonMass := 587.158, [5,14].SampleDuration := 927, [5,15].Run_ID := 2652, [5,15].Carbon_VOL_ml := 150.78236, [5,15].Carbon_MASS := 75.39118, [5,15].Carbon_DIST := 4.3399167, [5,15].Hour := 12, [5,15].Min := 28, [5,15].Day := 20, [5,15].Month := 11, [5,15].Year := 2021, [5,15].Sample_DO := 5.57177, [5,15].Sample_pH := 9.072857, [5,15].Sample_VOL := 17.371574, [5,15].Density := 409.96295, [5,15].EmptyDist := 1410.0, [5,15].FullDist := 1352.9304, [5,15].Carbon_mLperL := 8.679833, [5,15].Slurry_Weight := -10.52187, [5,15].Sample_Tank := 5, [5,15].Carbon_Height := 57.06958, [5,15].Sample_FlowRate := 1.2063593, [5,15].Sample_FillTime := 14.400001, [5,15].DisplacedCarbonVol := 1047.0997, [5,15].DisplacedCarbonMass := 523.54987, [5,15].SampleDuration := 931, [5,16].Run_ID := 2642, [5,16].Carbon_VOL_ml := 228.1006, [5,16].Carbon_MASS := 114.0503, [5,16].Carbon_DIST := 6.6439276, [5,16].Hour := 9, [5,16].Min := 55, [5,16].Day := 20, [5,16].Month := 11, [5,16].Year := 2021, [5,16].Sample_DO := 5.4806933, [5,16].Sample_pH := 9.119755, [5,16].Sample_VOL := 17.166096, [5,16].Density := 406.94293, [5,16].EmptyDist := 1410.0, [5,16].FullDist := 1323.6663, [5,16].Carbon_mLperL := 13.287855, [5,16].Slurry_Weight := -10.52187, [5,16].Sample_Tank := 5, [5,16].Carbon_Height := 86.33374, [5,16].Sample_FlowRate := 1.1003907, [5,16].Sample_FillTime := 15.600001, [5,16].DisplacedCarbonVol := 1462.1831, [5,16].DisplacedCarbonMass := 731.09155, [5,16].SampleDuration := 931, [5,17].Run_ID := 2633, [5,17].Carbon_VOL_ml := 219.35, [5,17].Carbon_MASS := 109.675, [5,17].Carbon_DIST := 6.2732816, [5,17].Hour := 7, [5,17].Min := 38,
        [5,17].Day := 20, [5,17].Month := 11, [5,17].Year := 2021, [5,17].Sample_DO := 6.0118947, [5,17].Sample_pH := 9.130824, [5,17].Sample_VOL := 17.482876, [5,17].Density := 411.5988, [5,17].EmptyDist := 1410.0, [5,17].FullDist := 1326.9783, [5,17].ErrorFlag := 1, [5,17].Carbon_mLperL := 12.546563, [5,17].Slurry_Weight := -10.52187, [5,17].Sample_Tank := 5, [5,17].Carbon_Height := 83.02173, [5,17].Sample_FlowRate := 1.2539717, [5,17].Sample_FillTime := 13.942001, [5,17].DisplacedCarbonVol := 1573.3035, [5,17].DisplacedCarbonMass := 786.65173, [5,17].SampleDuration := 171, [5,18].Run_ID := 2632, [5,18].Carbon_VOL_ml := 295.61685, [5,18].Carbon_MASS := 147.80843, [5,18].Carbon_DIST := 8.710406, [5,18].Hour := 7, [5,18].Min := 26, [5,18].Day := 20, [5,18].Month := 11, [5,18].Year := 2021, [5,18].Sample_DO := 5.8112407, [5,18].Sample_pH := 9.173185, [5,18].Sample_VOL := 16.969177, [5,18].Density := 404.04868, [5,18].EmptyDist := 1410.0, [5,18].FullDist := 1298.112, [5,18].Carbon_mLperL := 17.420813, [5,18].Slurry_Weight := -10.52187, [5,18].Sample_Tank := 5, [5,18].Carbon_Height := 111.88794, [5,18].Sample_FlowRate := 1.1206694, [5,18].Sample_FillTime := 15.142001, [5,18].DisplacedCarbonVol := 1952.297, [5,18].DisplacedCarbonMass := 976.1485, [5,18].SampleDuration := 931, [5,19].Run_ID := 2623, [5,19].Carbon_VOL_ml := 148.33186, [5,19].Carbon_MASS := 74.16593, [5,19].Carbon_DIST := 4.2380533, [5,19].Hour := 4, [5,19].Min := 36, [5,19].Day := 20, [5,19].Month := 11, [5,19].Year := 2021, [5,19].Sample_DO := 5.468576, [5,19].Sample_pH := 9.128056, [5,19].Sample_VOL := 17.5, [5,19].Density := 411.85046, [5,19].EmptyDist := 1410.0, [5,19].FullDist := 1353.8579, [5,19].Carbon_mLperL := 8.476107, [5,19].Slurry_Weight := -10.52187,
        [5,19].Sample_Tank := 5, [5,19].Carbon_Height := 56.14209, [5,19].Sample_FlowRate := 1.3418187, [5,19].Sample_FillTime := 13.042001, [5,19].DisplacedCarbonVol := 1137.3398, [5,19].DisplacedCarbonMass := 568.6699, [5,19].SampleDuration := 928, [6,0].Run_ID := 2790, [6,0].Min := 3, [6,0].Day := 22, [6,0].Month := 11, [6,0].Year := 2021, [6,0].Sample_DO := 5.1891594, [6,0].Sample_pH := 9.087861, [6,0].Sample_VOL := 17.893835, [6,0].Density := 417.63882, [6,0].EmptyDist := 1410.0, [6,0].FullDist := 1445.206, [6,0].Slurry_Weight := -10.52187, [6,0].Sample_Tank := 6, [6,0].Carbon_Height := -35.206055, [6,0].Sample_FlowRate := 1.8639408, [6,0].Sample_FillTime := 9.600001, [6,0].SampleDuration := 716, [6,1].Run_ID := 2777, [6,1].Hour := 20, [6,1].Min := 45, [6,1].Day := 21, [6,1].Month := 11, [6,1].Year := 2021, [6,1].Sample_DO := 5.281458, [6,1].Sample_pH := 9.0882015, [6,1].Sample_VOL := 17.226028, [6,1].Density := 407.82376, [6,1].EmptyDist := 1410.0, [6,1].FullDist := 1447.1489, [6,1].ErrorFlag := 1, [6,1].Slurry_Weight := -10.52187, [6,1].Sample_Tank := 6, [6,1].Carbon_Height := -37.148926, [6,1].Sample_FlowRate := 1.7943777, [6,1].Sample_FillTime := 9.600001, [6,1].SampleDuration := 704, [6,2].Run_ID := 2776, [6,2].Hour := 20, [6,2].Min := 33, [6,2].Day := 21, [6,2].Month := 11, [6,2].Year := 2021, [6,2].Sample_DO := 5.310106, [6,2].Sample_pH := 9.077998, [6,2].Sample_VOL := 17.619864, [6,2].Density := 413.61212, [6,2].EmptyDist := 1410.0, [6,2].FullDist := 1447.1489, [6,2].Slurry_Weight := -10.52187, [6,2].Sample_Tank := 6, [6,2].Carbon_Height := -37.148926, [6,2].Sample_FlowRate := 1.8354023, [6,2].Sample_FillTime := 9.600001,
        [6,2].SampleDuration := 710, [6,3].Run_ID := 2754, [6,3].Carbon_VOL_ml := 4.682983, [6,3].Carbon_MASS := 2.3414915, [6,3].Carbon_DIST := 0.13386501, [6,3].Hour := 14, [6,3].Min := 35, [6,3].Day := 21, [6,3].Month := 11, [6,3].Year := 2021, [6,3].Sample_DO := 5.068293, [6,3].Sample_pH := 9.049427, [6,3].Sample_VOL := 17.491438, [6,3].Density := 411.7246, [6,3].EmptyDist := 1410.0, [6,3].FullDist := 1408.2275, [6,3].ErrorFlag := 1, [6,3].Carbon_mLperL := 0.26773003, [6,3].Slurry_Weight := -10.52187, [6,3].Sample_Tank := 6, [6,3].Carbon_Height := 1.7724609, [6,3].Sample_FlowRate := 1.7954668, [6,3].Sample_FillTime := 9.742001, [6,3].DisplacedCarbonVol := 48.070038, [6,3].DisplacedCarbonMass := 24.035019, [6,3].SampleDuration := 704, [6,4].Run_ID := 2753, [6,4].Carbon_VOL_ml := 4.4897933, [6,4].Carbon_MASS := 2.2448967, [6,4].Carbon_DIST := 0.12954739, [6,4].Hour := 14, [6,4].Min := 23, [6,4].Day := 21, [6,4].Month := 11, [6,4].Year := 2021, [6,4].Sample_DO := 5.051355, [6,4].Sample_pH := 9.060365, [6,4].Sample_VOL := 17.328768, [6,4].Density := 409.3338, [6,4].EmptyDist := 1410.0, [6,4].FullDist := 1408.3007, [6,4].Carbon_mLperL := 0.25909477, [6,4].Slurry_Weight := -10.52187, [6,4].Sample_Tank := 6, [6,4].Carbon_Height := 1.6993408, [6,4].Sample_FlowRate := 1.8352854, [6,4].Sample_FillTime := 9.442001, [6,4].DisplacedCarbonVol := 47.55129, [6,4].DisplacedCarbonMass := 23.775644, [6,4].SampleDuration := 709, [6,5].Run_ID := 2739, [6,5].Carbon_VOL_ml := 144.26361, [6,5].Carbon_MASS := 72.131805, [6,5].Carbon_DIST := 4.227293, [6,5].Hour := 10, [6,5].Min := 53, [6,5].Day := 21, [6,5].Month := 11, [6,5].Year := 2021, [6,5].Sample_DO := 5.231105,
        [6,5].Sample_pH := 9.089754, [6,5].Sample_VOL := 17.063356, [6,5].Density := 405.4329, [6,5].EmptyDist := 1410.0, [6,5].FullDist := 1355.3977, [6,5].ErrorFlag := 1, [6,5].Carbon_mLperL := 8.454586, [6,5].Slurry_Weight := -10.52187, [6,5].Sample_Tank := 6, [6,5].Carbon_Height := 54.602295, [6,5].Sample_FlowRate := 1.8071758, [6,5].Sample_FillTime := 9.442001, [6,5].DisplacedCarbonVol := 1527.8923, [6,5].DisplacedCarbonMass := 763.94617, [6,5].SampleDuration := 705, [6,6].Run_ID := 2738, [6,6].Carbon_VOL_ml := 157.28017, [6,6].Carbon_MASS := 78.64008, [6,6].Carbon_DIST := 4.4849424, [6,6].Hour := 10, [6,6].Min := 41, [6,6].Day := 21, [6,6].Month := 11, [6,6].Year := 2021, [6,6].Sample_DO := 5.2317286, [6,6].Sample_pH := 9.203178, [6,6].Sample_VOL := 17.534246, [6,6].Density := 412.35376, [6,6].EmptyDist := 1410.0, [6,6].FullDist := 1350.4711, [6,6].Carbon_mLperL := 8.969885, [6,6].Slurry_Weight := -10.52187, [6,6].Sample_Tank := 6, [6,6].Carbon_Height := 59.52893, [6,6].Sample_FlowRate := 1.8264837, [6,6].Sample_FillTime := 9.600001, [6,6].DisplacedCarbonVol := 1638.335, [6,6].DisplacedCarbonMass := 819.1675, [6,6].SampleDuration := 708, [6,7].Run_ID := 2727, [6,7].Carbon_VOL_ml := 106.01279, [6,7].Carbon_MASS := 53.006393, [6,7].Carbon_DIST := 2.982248, [6,7].Hour := 7, [6,7].Min := 54, [6,7].Day := 21, [6,7].Month := 11, [6,7].Year := 2021, [6,7].Sample_DO := 4.8922467, [6,7].Sample_pH := 9.109035, [6,7].Sample_VOL := 17.773972, [6,7].Density := 415.87714, [6,7].EmptyDist := 1410.0, [6,7].FullDist := 1369.8752, [6,7].Carbon_mLperL := 5.964496, [6,7].Slurry_Weight := -10.52187, [6,7].Sample_Tank := 6, [6,7].Carbon_Height := 40.124756, [6,7].Sample_FlowRate := 1.8824369, [6,7].Sample_FillTime := 9.442001,
        [6,7].DisplacedCarbonVol := 1122.7788, [6,7].DisplacedCarbonMass := 561.3894, [6,7].SampleDuration := 707, [6,8].Run_ID := 2717, [6,8].Carbon_VOL_ml := 128.04861, [6,8].Carbon_MASS := 64.02431, [6,8].Carbon_DIST := 3.5728805, [6,8].Hour := 4, [6,8].Min := 33, [6,8].Day := 21, [6,8].Month := 11, [6,8].Year := 2021, [6,8].Sample_DO := 5.3341846, [6,8].Sample_pH := 9.228728, [6,8].Sample_VOL := 17.919521, [6,8].Density := 418.0164, [6,8].EmptyDist := 1410.0, [6,8].FullDist := 1361.5349, [6,8].Carbon_mLperL := 7.145761, [6,8].Slurry_Weight := -10.52187, [6,8].Sample_Tank := 6, [6,8].Carbon_Height := 48.465088, [6,8].Sample_FlowRate := 1.8978521, [6,8].Sample_FillTime := 9.442001, [6,8].DisplacedCarbonVol := 1356.1597, [6,8].DisplacedCarbonMass := 678.07983, [6,8].SampleDuration := 707, [6,9].Run_ID := 2706, [6,9].Carbon_VOL_ml := 236.31065, [6,9].Carbon_MASS := 118.15533, [6,9].Carbon_DIST := 6.758346, [6,9].Hour := 1, [6,9].Min := 50, [6,9].Day := 21, [6,9].Month := 11, [6,9].Year := 2021, [6,9].Sample_DO := 5.0642967, [6,9].Sample_pH := 9.100977, [6,9].Sample_VOL := 17.482876, [6,9].Density := 411.5988, [6,9].EmptyDist := 1410.0, [6,9].FullDist := 1320.5588, [6,9].ErrorFlag := 1, [6,9].Carbon_mLperL := 13.516692, [6,9].Slurry_Weight := -10.52187, [6,9].Sample_Tank := 6, [6,9].Carbon_Height := 89.44116, [6,9].Sample_FlowRate := 1.8211327, [6,9].Sample_FillTime := 9.600001, [6,9].DisplacedCarbonVol := 2461.5688, [6,9].DisplacedCarbonMass := 1230.7844, [6,9].SampleDuration := 705, [6,10].Run_ID := 2705, [6,10].Carbon_VOL_ml := 254.94003, [6,10].Carbon_MASS := 127.47002, [6,10].Carbon_DIST := 7.5845633, [6,10].Hour := 1, [6,10].Min := 38, [6,10].Day := 21, [6,10].Month := 11,
        [6,10].Year := 2021, [6,10].Sample_DO := 5.403073, [6,10].Sample_pH := 9.177628, [6,10].Sample_VOL := 16.806507, [6,10].Density := 401.65787, [6,10].EmptyDist := 1410.0, [6,10].FullDist := 1313.5078, [6,10].Carbon_mLperL := 15.1691265, [6,10].Slurry_Weight := -10.52187, [6,10].Sample_Tank := 6, [6,10].Carbon_Height := 96.49219, [6,10].Sample_FlowRate := 1.7799729, [6,10].Sample_FillTime := 9.442001, [6,10].DisplacedCarbonVol := 2700.0635, [6,10].DisplacedCarbonMass := 1350.0317, [6,10].SampleDuration := 709, [6,11].Run_ID := 2693, [6,11].Carbon_VOL_ml := 99.325676, [6,11].Carbon_MASS := 49.662838, [6,11].Carbon_DIST := 2.803586, [6,11].Hour := 22, [6,11].Min := 37, [6,11].Day := 20, [6,11].Month := 11, [6,11].Year := 2021, [6,11].Sample_DO := 5.500787, [6,11].Sample_pH := 9.197981, [6,11].Sample_VOL := 17.71404, [6,11].Density := 414.99634, [6,11].EmptyDist := 1410.0, [6,11].FullDist := 1372.4062, [6,11].Carbon_mLperL := 5.607172, [6,11].Slurry_Weight := -10.52187, [6,11].Sample_Tank := 6, [6,11].Carbon_Height := 37.59375, [6,11].Sample_FlowRate := 1.8452123, [6,11].Sample_FillTime := 9.600001, [6,11].DisplacedCarbonVol := 1034.6422, [6,11].DisplacedCarbonMass := 517.3211, [6,11].SampleDuration := 707, [6,12].Run_ID := 2680, [6,12].Carbon_VOL_ml := 110.58999, [6,12].Carbon_MASS := 55.294994, [6,12].Carbon_DIST := 3.1830733, [6,12].Hour := 19, [6,12].Min := 21, [6,12].Day := 20, [6,12].Month := 11, [6,12].Year := 2021, [6,12].Sample_DO := 5.1221933, [6,12].Sample_pH := 9.235373, [6,12].Sample_VOL := 17.371574, [6,12].Density := 409.96295, [6,12].EmptyDist := 1410.0, [6,12].FullDist := 1368.1428, [6,12].Carbon_mLperL := 6.3661466, [6,12].Slurry_Weight := -10.52187, [6,12].Sample_Tank := 6, [6,12].Carbon_Height := 41.857178, [6,12].Sample_FlowRate := 1.8398191,
        [6,12].Sample_FillTime := 9.442001, [6,12].DisplacedCarbonVol := 1171.2559, [6,12].DisplacedCarbonMass := 585.6279, [6,12].SampleDuration := 707, [6,13].Run_ID := 2667, [6,13].Carbon_VOL_ml := 204.08128, [6,13].Carbon_MASS := 102.04064, [6,13].Carbon_DIST := 5.876897, [6,13].Hour := 16, [6,13].Min := 7, [6,13].Day := 20, [6,13].Month := 11, [6,13].Year := 2021, [6,13].Sample_DO := 5.0148935, [6,13].Sample_pH := 9.118451, [6,13].Sample_VOL := 17.363014, [6,13].Density := 409.8371, [6,13].EmptyDist := 1410.0, [6,13].FullDist := 1332.7573, [6,13].ErrorFlag := 1, [6,13].Carbon_mLperL := 11.753794, [6,13].Slurry_Weight := -10.52187, [6,13].Sample_Tank := 6, [6,13].Carbon_Height := 77.242676, [6,13].Sample_FlowRate := 1.7538397, [6,13].Sample_FillTime := 9.900001, [6,13].DisplacedCarbonVol := 2061.427, [6,13].DisplacedCarbonMass := 1030.7135, [6,13].SampleDuration := 704, [6,14].Run_ID := 2666, [6,14].Carbon_VOL_ml := 205.96124, [6,14].Carbon_MASS := 102.98062, [6,14].Carbon_DIST := 5.744096, [6,14].Hour := 15, [6,14].Min := 56, [6,14].Day := 20, [6,14].Month := 11, [6,14].Year := 2021, [6,14].Sample_DO := 5.417887, [6,14].Sample_pH := 9.220958, [6,14].Sample_VOL := 17.928082, [6,14].Density := 418.14218, [6,14].EmptyDist := 1410.0, [6,14].FullDist := 1332.0458, [6,14].Carbon_mLperL := 11.488192, [6,14].Slurry_Weight := -10.52187, [6,14].Sample_Tank := 6, [6,14].Carbon_Height := 77.95422, [6,14].Sample_FlowRate := 1.7335216, [6,14].Sample_FillTime := 10.342001, [6,14].DisplacedCarbonVol := 1991.5028, [6,14].DisplacedCarbonMass := 995.7514, [6,14].SampleDuration := 708, [6,15].Run_ID := 2654, [6,15].Hour := 12, [6,15].Min := 51, [6,15].Day := 20, [6,15].Month := 11, [6,15].Year := 2021, [6,15].Sample_DO := 4.6927094,
        [6,15].Sample_pH := 9.046268, [6,15].Sample_VOL := 18.06507, [6,15].Density := 420.15552, [6,15].EmptyDist := 1410.0, [6,15].FullDist := 1430.4984, [6,15].ErrorFlag := 1, [6,15].Slurry_Weight := -10.52187, [6,15].Sample_Tank := 6, [6,15].Carbon_Height := -20.498413, [6,15].Sample_FlowRate := 1.8817778, [6,15].Sample_FillTime := 9.600001, [6,15].SampleDuration := 704, [6,16].Run_ID := 2653, [6,16].Carbon_VOL_ml := 128.82686, [6,16].Carbon_MASS := 64.41343, [6,16].Carbon_DIST := 3.6807673, [6,16].Hour := 12, [6,16].Min := 39, [6,16].Day := 20, [6,16].Month := 11, [6,16].Year := 2021, [6,16].Sample_DO := 4.8201733, [6,16].Sample_pH := 9.035338, [6,16].Sample_VOL := 17.5, [6,16].Density := 411.85046, [6,16].EmptyDist := 1410.0, [6,16].FullDist := 1361.2404, [6,16].Carbon_mLperL := 7.3615346, [6,16].Slurry_Weight := -10.52187, [6,16].Sample_Tank := 6, [6,16].Carbon_Height := 48.759644, [6,16].Sample_FlowRate := 1.8534206, [6,16].Sample_FillTime := 9.442001, [6,16].DisplacedCarbonVol := 1364.4021, [6,16].DisplacedCarbonMass := 682.20105, [6,16].SampleDuration := 708, [6,17].Run_ID := 2643, [6,17].Carbon_VOL_ml := 77.92522, [6,17].Carbon_MASS := 38.96261, [6,17].Carbon_DIST := 2.1974082, [6,17].Hour := 10, [6,17].Min := 7, [6,17].Day := 20, [6,17].Month := 11, [6,17].Year := 2021, [6,17].Sample_DO := 5.2950706, [6,17].Sample_pH := 9.183289, [6,17].Sample_VOL := 17.731165, [6,17].Density := 415.24802, [6,17].EmptyDist := 1410.0, [6,17].FullDist := 1380.5061, [6,17].Carbon_mLperL := 4.3948164, [6,17].Slurry_Weight := -10.52187, [6,17].Sample_Tank := 6, [6,17].Carbon_Height := 29.493896, [6,17].Sample_FlowRate := 1.7908456, [6,17].Sample_FillTime := 9.901001, [6,17].DisplacedCarbonVol := 787.04376, [6,17].DisplacedCarbonMass := 393.52188, [6,17].SampleDuration := 711,
        [6,18].Run_ID := 2634, [6,18].Carbon_VOL_ml := 124.58862, [6,18].Carbon_MASS := 62.29431, [6,18].Carbon_DIST := 3.5098774, [6,18].Hour := 7, [6,18].Min := 49, [6,18].Day := 20, [6,18].Month := 11, [6,18].Year := 2021, [6,18].Sample_DO := 5.131065, [6,18].Sample_pH := 9.112165, [6,18].Sample_VOL := 17.748287, [6,18].Density := 415.49963, [6,18].EmptyDist := 1410.0, [6,18].FullDist := 1362.8445, [6,18].Carbon_mLperL := 7.019755, [6,18].Slurry_Weight := -10.52187, [6,18].Sample_Tank := 6, [6,18].Carbon_Height := 47.155518, [6,18].Sample_FlowRate := 1.8487797, [6,18].Sample_FillTime := 9.600001, [6,18].DisplacedCarbonVol := 1297.7981, [6,18].DisplacedCarbonMass := 648.89905, [6,18].SampleDuration := 709, [6,19].Run_ID := 2624, [6,19].Carbon_VOL_ml := 198.76553, [6,19].Carbon_MASS := 99.38277, [6,19].Carbon_DIST := 5.684578, [6,19].Hour := 4, [6,19].Min := 47, [6,19].Day := 20, [6,19].Month := 11, [6,19].Year := 2021, [6,19].Sample_DO := 5.013442, [6,19].Sample_pH := 9.131547, [6,19].Sample_VOL := 17.482876, [6,19].Density := 411.5988, [6,19].EmptyDist := 1410.0, [6,19].FullDist := 1334.7693, [6,19].Carbon_mLperL := 11.369156, [6,19].Slurry_Weight := -10.52187, [6,19].Sample_Tank := 6, [6,19].Carbon_Height := 75.23071, [6,19].Sample_FlowRate := 1.8484747, [6,19].Sample_FillTime := 9.458001, [6,19].DisplacedCarbonVol := 2101.5598, [6,19].DisplacedCarbonMass := 1050.7799, [6,19].SampleDuration := 709, [7,0].Run_ID := 2779, [7,0].Hour := 21, [7,0].Min := 19, [7,0].Day := 21, [7,0].Month := 11, [7,0].Year := 2021, [7,0].Sample_DO := 5.578247, [7,0].Sample_pH := 9.083747, [7,0].Sample_VOL := 17.388699, [7,0].Density := 410.2146, [7,0].EmptyDist := 1410.0, [7,0].FullDist := 1445.2788,
        [7,0].ErrorFlag := 1, [7,0].Slurry_Weight := -10.52187, [7,0].Sample_Tank := 7, [7,0].Carbon_Height := -35.27881, [7,0].Sample_FlowRate := 1.7047743, [7,0].Sample_FillTime := 10.200001, [7,0].SampleDuration := 1025, [7,1].Run_ID := 2778, [7,1].Hour := 21, [7,1].Min := 2, [7,1].Day := 21, [7,1].Month := 11, [7,1].Year := 2021, [7,1].Sample_DO := 5.4229026, [7,1].Sample_pH := 9.10397, [7,1].Sample_VOL := 16.489727, [7,1].Density := 397.002, [7,1].EmptyDist := 1410.0, [7,1].FullDist := 1445.1282, [7,1].Slurry_Weight := -10.52187, [7,1].Sample_Tank := 7, [7,1].Carbon_Height := -35.128174, [7,1].Sample_FlowRate := 1.7176796, [7,1].Sample_FillTime := 9.600001, [7,1].SampleDuration := 704, [7,2].Run_ID := 2765, [7,2].Hour := 17, [7,2].Min := 50, [7,2].Day := 21, [7,2].Month := 11, [7,2].Year := 2021, [7,2].Sample_DO := 5.2878976, [7,2].Sample_pH := 9.129586, [7,2].Sample_VOL := 17.508562, [7,2].Density := 411.9763, [7,2].EmptyDist := 1410.0, [7,2].FullDist := 1447.0637, [7,2].ErrorFlag := 1, [7,2].Slurry_Weight := -10.52187, [7,2].Sample_Tank := 7, [7,2].Carbon_Height := -37.06372, [7,2].Sample_FlowRate := 1.7685416, [7,2].Sample_FillTime := 9.900001, [7,2].SampleDuration := 1181, [7,3].Run_ID := 2764, [7,3].Hour := 17, [7,3].Min := 33, [7,3].Day := 21, [7,3].Month := 11, [7,3].Year := 2021, [7,3].Sample_DO := 5.6656094, [7,3].Sample_pH := 9.232738, [7,3].Sample_VOL := 17.722603, [7,3].Density := 415.12213, [7,3].EmptyDist := 1410.0, [7,3].FullDist := 1447.073, [7,3].Slurry_Weight := -10.52187, [7,3].Sample_Tank := 7, [7,3].Carbon_Height := -37.072998, [7,3].Sample_FlowRate := 1.7136532,
        [7,3].Sample_FillTime := 10.342001, [7,3].SampleDuration := 781, [7,4].Run_ID := 2756, [7,4].Hour := 15, [7,4].Min := 9, [7,4].Day := 21, [7,4].Month := 11, [7,4].Year := 2021, [7,4].Sample_DO := 5.035901, [7,4].Sample_pH := 9.089533, [7,4].Sample_VOL := 17.388699, [7,4].Density := 410.2146, [7,4].EmptyDist := 1410.0, [7,4].FullDist := 1446.8662, [7,4].ErrorFlag := 1, [7,4].Slurry_Weight := -10.52187, [7,4].Sample_Tank := 7, [7,4].Carbon_Height := -36.86621, [7,4].Sample_FlowRate := 1.6813669, [7,4].Sample_FillTime := 10.342001, [7,4].SampleDuration := 1024, [7,5].Run_ID := 2755, [7,5].Carbon_VOL_ml := 47.627094, [7,5].Carbon_MASS := 23.813547, [7,5].Carbon_DIST := 1.384481, [7,5].Hour := 14, [7,5].Min := 52, [7,5].Day := 21, [7,5].Month := 11, [7,5].Year := 2021, [7,5].Sample_DO := 5.2279263, [7,5].Sample_pH := 9.131461, [7,5].Sample_VOL := 17.200342, [7,5].Density := 407.44623, [7,5].EmptyDist := 1410.0, [7,5].FullDist := 1391.9736, [7,5].Carbon_mLperL := 2.768962, [7,5].Slurry_Weight := -10.52187, [7,5].Sample_Tank := 7, [7,5].Carbon_Height := 18.026367, [7,5].Sample_FlowRate := 1.6631542, [7,5].Sample_FillTime := 10.342001, [7,5].DisplacedCarbonVol := 460.5211, [7,5].DisplacedCarbonMass := 230.26054, [7,5].SampleDuration := 704, [7,6].Run_ID := 2741, [7,6].Carbon_VOL_ml := 217.16817, [7,6].Carbon_MASS := 108.58408, [7,6].Carbon_DIST := 6.2017703, [7,6].Hour := 11, [7,6].Min := 27, [7,6].Day := 21, [7,6].Month := 11, [7,6].Year := 2021, [7,6].Sample_DO := 5.2502227, [7,6].Sample_pH := 9.080902, [7,6].Sample_VOL := 17.508562, [7,6].Density := 411.9763, [7,6].EmptyDist := 1410.0, [7,6].FullDist := 1327.8041,
        [7,6].ErrorFlag := 1, [7,6].Carbon_mLperL := 12.403541, [7,6].Slurry_Weight := -10.52187, [7,6].Sample_Tank := 7, [7,6].Carbon_Height := 82.19592, [7,6].Sample_FlowRate := 1.7685416, [7,6].Sample_FillTime := 9.900001, [7,6].DisplacedCarbonVol := 2193.618, [7,6].DisplacedCarbonMass := 1096.809, [7,6].SampleDuration := 1025, [7,7].Run_ID := 2740, [7,7].Carbon_VOL_ml := 168.70349, [7,7].Carbon_MASS := 84.351746, [7,7].Carbon_DIST := 4.867729, [7,7].Hour := 11, [7,7].Min := 10, [7,7].Day := 21, [7,7].Month := 11, [7,7].Year := 2021, [7,7].Sample_DO := 5.156539, [7,7].Sample_pH := 9.155446, [7,7].Sample_VOL := 17.328768, [7,7].Density := 409.3338, [7,7].EmptyDist := 1410.0, [7,7].FullDist := 1346.1475, [7,7].Carbon_mLperL := 9.735458, [7,7].Slurry_Weight := -10.52187, [7,7].Sample_Tank := 7, [7,7].Carbon_Height := 63.85254, [7,7].Sample_FlowRate := 1.7503805, [7,7].Sample_FillTime := 9.900001, [7,7].DisplacedCarbonVol := 1704.0757, [7,7].DisplacedCarbonMass := 852.03784, [7,7].SampleDuration := 705, [7,8].Run_ID := 2728, [7,8].Carbon_VOL_ml := 101.72329, [7,8].Carbon_MASS := 50.861645, [7,8].Carbon_DIST := 3.0155535, [7,8].Hour := 8, [7,8].Min := 11, [7,8].Day := 21, [7,8].Month := 11, [7,8].Year := 2021, [7,8].Sample_DO := 5.2242136, [7,8].Sample_pH := 9.224625, [7,8].Sample_VOL := 16.866438, [7,8].Density := 402.5387, [7,8].EmptyDist := 1410.0, [7,8].FullDist := 1371.4988, [7,8].Carbon_mLperL := 6.031107, [7,8].Slurry_Weight := -10.52187, [7,8].Sample_Tank := 7, [7,8].Carbon_Height := 38.50122, [7,8].Sample_FlowRate := 1.8417162, [7,8].Sample_FillTime := 9.158001, [7,8].DisplacedCarbonVol := 1110.7587, [7,8].DisplacedCarbonMass := 555.37933, [7,8].SampleDuration := 794, [7,9].Run_ID := 2718, [7,9].Carbon_VOL_ml := 160.73466,
        [7,9].Carbon_MASS := 80.36733, [7,9].Carbon_DIST := 4.665459, [7,9].Hour := 4, [7,9].Min := 50, [7,9].Day := 21, [7,9].Month := 11, [7,9].Year := 2021, [7,9].Sample_DO := 5.3953185, [7,9].Sample_pH := 9.24873, [7,9].Sample_VOL := 17.226028, [7,9].Density := 407.82376, [7,9].EmptyDist := 1410.0, [7,9].FullDist := 1349.1636, [7,9].Carbon_mLperL := 9.330918, [7,9].Slurry_Weight := -10.52187, [7,9].Sample_Tank := 7, [7,9].Carbon_Height := 60.836426, [7,9].Sample_FlowRate := 1.7400028, [7,9].Sample_FillTime := 9.900001, [7,9].DisplacedCarbonVol := 1623.5825, [7,9].DisplacedCarbonMass := 811.79126, [7,9].SampleDuration := 703, [7,10].Run_ID := 2707, [7,10].Carbon_VOL_ml := 119.72116, [7,10].Carbon_MASS := 59.86058, [7,10].Carbon_DIST := 3.4819303, [7,10].Hour := 2, [7,10].Min := 7, [7,10].Day := 21, [7,10].Month := 11, [7,10].Year := 2021, [7,10].Sample_DO := 4.987476, [7,10].Sample_pH := 9.1145115, [7,10].Sample_VOL := 17.19178, [7,10].Density := 407.3204, [7,10].EmptyDist := 1410.0, [7,10].FullDist := 1364.6868, [7,10].Carbon_mLperL := 6.9638605, [7,10].Slurry_Weight := -10.52187, [7,10].Sample_Tank := 7, [7,10].Carbon_Height := 45.313232, [7,10].Sample_FlowRate := 1.7365433, [7,10].Sample_FillTime := 9.900001, [7,10].DisplacedCarbonVol := 1209.3046, [7,10].DisplacedCarbonMass := 604.6523, [7,10].SampleDuration := 705, [7,11].Run_ID := 2694, [7,11].Carbon_VOL_ml := 191.82812, [7,11].Carbon_MASS := 95.91406, [7,11].Carbon_DIST := 5.567973, [7,11].Hour := 22, [7,11].Min := 54, [7,11].Day := 20, [7,11].Month := 11, [7,11].Year := 2021, [7,11].Sample_DO := 5.077548, [7,11].Sample_pH := 9.136234, [7,11].Sample_VOL := 17.226028, [7,11].Density := 407.82376, [7,11].EmptyDist := 1410.0,
        [7,11].FullDist := 1337.395, [7,11].Carbon_mLperL := 11.135946, [7,11].Slurry_Weight := -10.52187, [7,11].Sample_Tank := 7, [7,11].Carbon_Height := 72.60498, [7,11].Sample_FlowRate := 1.7400028, [7,11].Sample_FillTime := 9.900001, [7,11].DisplacedCarbonVol := 1937.6578, [7,11].DisplacedCarbonMass := 968.8289, [7,11].SampleDuration := 704, [7,12].Run_ID := 2682, [7,12].Carbon_VOL_ml := 154.25526, [7,12].Carbon_MASS := 77.12763, [7,12].Carbon_DIST := 4.457451, [7,12].Hour := 19, [7,12].Min := 55, [7,12].Day := 20, [7,12].Month := 11, [7,12].Year := 2021, [7,12].Sample_DO := 4.870401, [7,12].Sample_pH := 9.148639, [7,12].Sample_VOL := 17.303082, [7,12].Density := 408.95624, [7,12].EmptyDist := 1410.0, [7,12].FullDist := 1351.616, [7,12].ErrorFlag := 1, [7,12].Carbon_mLperL := 8.914902, [7,12].Slurry_Weight := -10.52187, [7,12].Sample_Tank := 7, [7,12].Carbon_Height := 58.384033, [7,12].Sample_FlowRate := 1.802404, [7,12].Sample_FillTime := 9.600001, [7,12].DisplacedCarbonVol := 1606.8254, [7,12].DisplacedCarbonMass := 803.4127, [7,12].SampleDuration := 1025, [7,13].Run_ID := 2681, [7,13].Carbon_VOL_ml := 193.97093, [7,13].Carbon_MASS := 96.985466, [7,13].Carbon_DIST := 5.32827, [7,13].Hour := 19, [7,13].Min := 38, [7,13].Day := 20, [7,13].Month := 11, [7,13].Year := 2021, [7,13].Sample_DO := 5.0747023, [7,13].Sample_pH := 9.267177, [7,13].Sample_VOL := 18.202055, [7,13].Density := 422.16888, [7,13].EmptyDist := 1410.0, [7,13].FullDist := 1336.584, [7,13].Carbon_mLperL := 10.65654, [7,13].Slurry_Weight := -10.52187, [7,13].Sample_Tank := 7, [7,13].Carbon_Height := 73.416016, [7,13].Sample_FlowRate := 1.8125925, [7,13].Sample_FillTime := 10.042001, [7,13].DisplacedCarbonVol := 1931.5966, [7,13].DisplacedCarbonMass := 965.7983, [7,13].SampleDuration := 704, [7,14].Run_ID := 2669,
        [7,14].Carbon_VOL_ml := 52.508427, [7,14].Carbon_MASS := 26.254213, [7,14].Carbon_DIST := 1.4721518, [7,14].Hour := 16, [7,14].Min := 41, [7,14].Day := 20, [7,14].Month := 11, [7,14].Year := 2021, [7,14].Sample_DO := 5.0697193, [7,14].Sample_pH := 9.191299, [7,14].Sample_VOL := 17.833904, [7,14].Density := 416.75797, [7,14].EmptyDist := 1410.0, [7,14].FullDist := 1390.1261, [7,14].ErrorFlag := 1, [7,14].Carbon_mLperL := 2.9443035, [7,14].Slurry_Weight := -10.52187, [7,14].Sample_Tank := 7, [7,14].Carbon_Height := 19.873901, [7,14].Sample_FlowRate := 1.7484219, [7,14].Sample_FillTime := 10.200001, [7,14].DisplacedCarbonVol := 514.7885, [7,14].DisplacedCarbonMass := 257.39426, [7,14].SampleDuration := 1024, [7,15].Run_ID := 2668, [7,15].Carbon_VOL_ml := 43.655914, [7,15].Carbon_MASS := 21.827957, [7,15].Carbon_DIST := 1.242449, [7,15].Hour := 16, [7,15].Min := 24, [7,15].Day := 20, [7,15].Month := 11, [7,15].Year := 2021, [7,15].Sample_DO := 5.207411, [7,15].Sample_pH := 9.140305, [7,15].Sample_VOL := 17.568493, [7,15].Density := 412.85712, [7,15].EmptyDist := 1410.0, [7,15].FullDist := 1393.4767, [7,15].Carbon_mLperL := 2.484898, [7,15].Slurry_Weight := -10.52187, [7,15].Sample_Tank := 7, [7,15].Carbon_Height := 16.523315, [7,15].Sample_FlowRate := 1.6987518, [7,15].Sample_FillTime := 10.342001, [7,15].DisplacedCarbonVol := 422.12253, [7,15].DisplacedCarbonMass := 211.06126, [7,15].SampleDuration := 704, [7,16].Run_ID := 2656, [7,16].Carbon_VOL_ml := 94.01443, [7,16].Carbon_MASS := 47.007214, [7,16].Carbon_DIST := 2.6207364, [7,16].Hour := 13, [7,16].Min := 25, [7,16].Day := 20, [7,16].Month := 11, [7,16].Year := 2021, [7,16].Sample_DO := 4.7953486, [7,16].Sample_pH := 9.043981, [7,16].Sample_VOL := 17.936644,
        [7,16].Density := 418.268, [7,16].EmptyDist := 1410.0, [7,16].FullDist := 1374.4165, [7,16].ErrorFlag := 1, [7,16].Carbon_mLperL := 5.2414727, [7,16].Slurry_Weight := -10.52187, [7,16].Sample_Tank := 7, [7,16].Carbon_Height := 35.583496, [7,16].Sample_FlowRate := 1.7861624, [7,16].Sample_FillTime := 10.042001, [7,16].DisplacedCarbonVol := 936.21216, [7,16].DisplacedCarbonMass := 468.10608, [7,16].SampleDuration := 1026, [7,17].Run_ID := 2655, [7,17].Hour := 13, [7,17].Min := 8, [7,17].Day := 20, [7,17].Month := 11, [7,17].Year := 2021, [7,17].Sample_DO := 5.0981183, [7,17].Sample_pH := 9.105702, [7,17].Sample_VOL := 17.234589, [7,17].Density := 407.94955, [7,17].EmptyDist := 1410.0, [7,17].FullDist := 1429.6099, [7,17].Slurry_Weight := -10.52187, [7,17].Sample_Tank := 7, [7,17].Carbon_Height := -19.609863, [7,17].Sample_FlowRate := 1.7408675, [7,17].Sample_FillTime := 9.900001, [7,17].SampleDuration := 705, [7,18].Run_ID := 2645, [7,18].Carbon_VOL_ml := 142.91934, [7,18].Carbon_MASS := 71.45967, [7,18].Carbon_DIST := 4.010807, [7,18].Hour := 10, [7,18].Min := 41, [7,18].Day := 20, [7,18].Month := 11, [7,18].Year := 2021, [7,18].Sample_DO := 5.1748085, [7,18].Sample_pH := 9.064751, [7,18].Sample_VOL := 17.81678, [7,18].Density := 416.5063, [7,18].EmptyDist := 1410.0, [7,18].FullDist := 1355.9065, [7,18].ErrorFlag := 1, [7,18].Carbon_mLperL := 8.021614, [7,18].Slurry_Weight := -10.52187, [7,18].Sample_Tank := 7, [7,18].Carbon_Height := 54.093506, [7,18].Sample_FlowRate := 1.8559144, [7,18].Sample_FillTime := 9.600001, [7,18].DisplacedCarbonVol := 1488.7428, [7,18].DisplacedCarbonMass := 744.3714, [7,18].SampleDuration := 1025, [7,19].Run_ID := 2644, [7,19].Carbon_VOL_ml := 155.31989, [7,19].Carbon_MASS := 77.65994, [7,19].Carbon_DIST := 4.567312,
        [7,19].Hour := 10, [7,19].Min := 24, [7,19].Day := 20, [7,19].Month := 11, [7,19].Year := 2021, [7,19].Sample_DO := 4.977071, [7,19].Sample_pH := 9.090282, [7,19].Sample_VOL := 17.003426, [7,19].Density := 404.55206, [7,19].EmptyDist := 1410.0, [7,19].FullDist := 1351.213, [7,19].Carbon_mLperL := 9.134624, [7,19].Slurry_Weight := -10.52187, [7,19].Sample_Tank := 7, [7,19].Carbon_Height := 58.786987, [7,19].Sample_FlowRate := 1.7175176, [7,19].Sample_FillTime := 9.900001, [7,19].DisplacedCarbonVol := 1568.8876, [7,19].DisplacedCarbonMass := 784.4438, [7,19].SampleDuration := 705, [8,0].Run_ID := 2781, [8,0].Hour := 21, [8,0].Min := 52, [8,0].Day := 21, [8,0].Month := 11, [8,0].Year := 2021, [8,0].Sample_DO := 5.314984, [8,0].Sample_pH := 9.142456, [8,0].Sample_VOL := 17.465754, [8,0].Density := 411.34714, [8,0].EmptyDist := 1410.0, [8,0].FullDist := 1447.225, [8,0].ErrorFlag := 1, [8,0].Slurry_Weight := -10.52187, [8,0].Sample_Tank := 8, [8,0].Carbon_Height := -37.224976, [8,0].Sample_FlowRate := 2.0792563, [8,0].Sample_FillTime := 8.400001, [8,0].SampleDuration := 974, [8,1].Run_ID := 2780, [8,1].Hour := 21, [8,1].Min := 36, [8,1].Day := 21, [8,1].Month := 11, [8,1].Year := 2021, [8,1].Sample_DO := 5.18206, [8,1].Sample_pH := 9.196667, [8,1].Sample_VOL := 17.328768, [8,1].Density := 409.3338, [8,1].EmptyDist := 1410.0, [8,1].FullDist := 1447.2201, [8,1].Slurry_Weight := -10.52187, [8,1].Sample_Tank := 8, [8,1].Carbon_Height := -37.220093, [8,1].Sample_FlowRate := 2.0629485, [8,1].Sample_FillTime := 8.400001, [8,1].SampleDuration := 1025, [8,2].Run_ID := 2767, [8,2].Hour := 18, [8,2].Min := 23,
        [8,2].Day := 21, [8,2].Month := 11, [8,2].Year := 2021, [8,2].Sample_DO := 5.147652, [8,2].Sample_pH := 9.237636, [8,2].Sample_VOL := 17.020548, [8,2].Density := 404.8037, [8,2].EmptyDist := 1410.0, [8,2].FullDist := 1447.1489, [8,2].ErrorFlag := 1, [8,2].Slurry_Weight := -10.52187, [8,2].Sample_Tank := 8, [8,2].Carbon_Height := -37.148926, [8,2].Sample_FlowRate := 2.0610976, [8,2].Sample_FillTime := 8.258001, [8,2].SampleDuration := 974, [8,3].Run_ID := 2766, [8,3].Hour := 18, [8,3].Min := 7, [8,3].Day := 21, [8,3].Month := 11, [8,3].Year := 2021, [8,3].Sample_DO := 5.0724254, [8,3].Sample_pH := 9.212067, [8,3].Sample_VOL := 18.030823, [8,3].Density := 419.65216, [8,3].EmptyDist := 1410.0, [8,3].FullDist := 1446.686, [8,3].Slurry_Weight := -10.52187, [8,3].Sample_Tank := 8, [8,3].Carbon_Height := -36.686035, [8,3].Sample_FlowRate := 2.072508, [8,3].Sample_FillTime := 8.700001, [8,3].SampleDuration := 1024, [8,4].Run_ID := 2758, [8,4].Hour := 15, [8,4].Min := 41, [8,4].Day := 21, [8,4].Month := 11, [8,4].Year := 2021, [8,4].Sample_DO := 4.6467757, [8,4].Sample_pH := 9.19162, [8,4].Sample_VOL := 16.738014, [8,4].Density := 400.65118, [8,4].EmptyDist := 1410.0, [8,4].FullDist := 1445.3447, [8,4].ErrorFlag := 1, [8,4].Slurry_Weight := -10.52187, [8,4].Sample_Tank := 8, [8,4].Carbon_Height := -35.344727, [8,4].Sample_FlowRate := 2.107531, [8,4].Sample_FillTime := 7.942001, [8,4].SampleDuration := 974, [8,5].Run_ID := 2757, [8,5].Hour := 15, [8,5].Min := 25, [8,5].Day := 21, [8,5].Month := 11, [8,5].Year := 2021, [8,5].Sample_DO := 4.830787,
        [8,5].Sample_pH := 9.186548, [8,5].Sample_VOL := 16.50685, [8,5].Density := 397.25366, [8,5].EmptyDist := 1410.0, [8,5].FullDist := 1436.9912, [8,5].Slurry_Weight := -10.52187, [8,5].Sample_Tank := 8, [8,5].Carbon_Height := -26.99121, [8,5].Sample_FlowRate := 2.0784245, [8,5].Sample_FillTime := 7.942001, [8,5].SampleDuration := 1026, [8,6].Run_ID := 2742, [8,6].Carbon_VOL_ml := 170.42476, [8,6].Carbon_MASS := 85.21238, [8,6].Carbon_DIST := 4.9467225, [8,6].Hour := 11, [8,6].Min := 43, [8,6].Day := 21, [8,6].Month := 11, [8,6].Year := 2021, [8,6].Sample_DO := 4.8775206, [8,6].Sample_pH := 9.193978, [8,6].Sample_VOL := 17.226028, [8,6].Density := 407.82376, [8,6].EmptyDist := 1410.0, [8,6].FullDist := 1345.496, [8,6].Carbon_mLperL := 9.893445, [8,6].Slurry_Weight := -10.52187, [8,6].Sample_Tank := 8, [8,6].Carbon_Height := 64.50403, [8,6].Sample_FlowRate := 2.2084649, [8,6].Sample_FillTime := 7.800001, [8,6].DisplacedCarbonVol := 1747.946, [8,6].DisplacedCarbonMass := 873.973, [8,6].SampleDuration := 1025, [8,7].Run_ID := 2729, [8,7].Carbon_VOL_ml := 329.18982, [8,7].Carbon_MASS := 164.59491, [8,7].Carbon_DIST := 9.255987, [8,7].Hour := 8, [8,7].Min := 27, [8,7].Day := 21, [8,7].Month := 11, [8,7].Year := 2021, [8,7].Sample_DO := 5.0847483, [8,7].Sample_pH := 9.237854, [8,7].Sample_VOL := 17.782534, [8,7].Density := 416.003, [8,7].EmptyDist := 1410.0, [8,7].FullDist := 1285.405, [8,7].Carbon_mLperL := 18.511974, [8,7].Slurry_Weight := -10.52187, [8,7].Sample_Tank := 8, [8,7].Carbon_Height := 124.59497, [8,7].Sample_FlowRate := 2.1575506, [8,7].Sample_FillTime := 8.242001, [8,7].DisplacedCarbonVol := 3195.2417, [8,7].DisplacedCarbonMass := 1597.6208, [8,7].SampleDuration := 1023, [8,8].Run_ID := 2719,
        [8,8].Carbon_VOL_ml := 295.60394, [8,8].Carbon_MASS := 147.80197, [8,8].Carbon_DIST := 8.926199, [8,8].Hour := 5, [8,8].Min := 7, [8,8].Day := 21, [8,8].Month := 11, [8,8].Year := 2021, [8,8].Sample_DO := 4.7715683, [8,8].Sample_pH := 9.265624, [8,8].Sample_VOL := 16.55822, [8,8].Density := 398.00867, [8,8].EmptyDist := 1410.0, [8,8].FullDist := 1298.117, [8,8].Carbon_mLperL := 17.852398, [8,8].Slurry_Weight := -10.52187, [8,8].Sample_Tank := 8, [8,8].Carbon_Height := 111.88306, [8,8].Sample_FlowRate := 2.2503693, [8,8].Sample_FillTime := 7.3580008, [8,8].DisplacedCarbonVol := 3213.959, [8,8].DisplacedCarbonMass := 1606.9795, [8,8].SampleDuration := 1023, [8,9].Run_ID := 2708, [8,9].Carbon_VOL_ml := 300.86197, [8,9].Carbon_MASS := 150.43098, [8,9].Carbon_DIST := 8.570897, [8,9].Hour := 2, [8,9].Min := 23, [8,9].Day := 21, [8,9].Month := 11, [8,9].Year := 2021, [8,9].Sample_DO := 4.822002, [8,9].Sample_pH := 9.214813, [8,9].Sample_VOL := 17.55137, [8,9].Density := 412.60544, [8,9].EmptyDist := 1410.0, [8,9].FullDist := 1296.1268, [8,9].Carbon_mLperL := 17.141794, [8,9].Slurry_Weight := -10.52187, [8,9].Sample_Tank := 8, [8,9].Carbon_Height := 113.87317, [8,9].Sample_FlowRate := 2.2501755, [8,9].Sample_FillTime := 7.800001, [8,9].DisplacedCarbonVol := 3085.7637, [8,9].DisplacedCarbonMass := 1542.8818, [8,9].SampleDuration := 1024, [8,10].Run_ID := 2695, [8,10].Carbon_VOL_ml := 217.18849, [8,10].Carbon_MASS := 108.594246, [8,10].Carbon_DIST := 6.448301, [8,10].Hour := 23, [8,10].Min := 11, [8,10].Day := 20, [8,10].Month := 11, [8,10].Year := 2021, [8,10].Sample_DO := 5.254755, [8,10].Sample_pH := 9.229914, [8,10].Sample_VOL := 16.840754, [8,10].Density := 402.16122,
        [8,10].EmptyDist := 1410.0, [8,10].FullDist := 1327.7964, [8,10].Carbon_mLperL := 12.896602, [8,10].Slurry_Weight := -10.52187, [8,10].Sample_Tank := 8, [8,10].Carbon_Height := 82.20361, [8,10].Sample_FlowRate := 2.1590707, [8,10].Sample_FillTime := 7.800001, [8,10].DisplacedCarbonVol := 2227.574, [8,10].DisplacedCarbonMass := 1113.787, [8,10].SampleDuration := 1025, [8,11].Run_ID := 2683, [8,11].Carbon_VOL_ml := 257.40988, [8,11].Carbon_MASS := 128.70494, [8,11].Carbon_DIST := 7.7249417, [8,11].Hour := 20, [8,11].Min := 11, [8,11].Day := 20, [8,11].Month := 11, [8,11].Year := 2021, [8,11].Sample_DO := 5.0393424, [8,11].Sample_pH := 9.250666, [8,11].Sample_VOL := 16.66096, [8,11].Density := 399.51865, [8,11].EmptyDist := 1410.0, [8,11].FullDist := 1312.573, [8,11].Carbon_mLperL := 15.449883, [8,11].Slurry_Weight := -10.52187, [8,11].Sample_Tank := 8, [8,11].Carbon_Height := 97.427, [8,11].Sample_FlowRate := 2.221461, [8,11].Sample_FillTime := 7.500001, [8,11].DisplacedCarbonVol := 2745.7053, [8,11].DisplacedCarbonMass := 1372.8527, [8,11].SampleDuration := 1023, [8,12].Run_ID := 2670, [8,12].Carbon_VOL_ml := 290.43362, [8,12].Carbon_MASS := 145.21681, [8,12].Carbon_DIST := 8.724961, [8,12].Hour := 16, [8,12].Min := 58, [8,12].Day := 20, [8,12].Month := 11, [8,12].Year := 2021, [8,12].Sample_DO := 4.5596857, [8,12].Sample_pH := 9.233557, [8,12].Sample_VOL := 16.643835, [8,12].Density := 399.26697, [8,12].EmptyDist := 1410.0, [8,12].FullDist := 1300.0739, [8,12].Carbon_mLperL := 17.449923, [8,12].Slurry_Weight := -10.52187, [8,12].Sample_Tank := 8, [8,12].Carbon_Height := 109.92615, [8,12].Sample_FlowRate := 2.2191777, [8,12].Sample_FillTime := 7.500001, [8,12].DisplacedCarbonVol := 3097.9585, [8,12].DisplacedCarbonMass := 1548.9792, [8,12].SampleDuration := 1025, [8,13].Run_ID := 2657,
        [8,13].Carbon_VOL_ml := 353.2772, [8,13].Carbon_MASS := 176.6386, [8,13].Carbon_DIST := 10.054283, [8,13].Hour := 13, [8,13].Min := 41, [8,13].Day := 20, [8,13].Month := 11, [8,13].Year := 2021, [8,13].Sample_DO := 4.9041905, [8,13].Sample_pH := 9.174795, [8,13].Sample_VOL := 17.568493, [8,13].Density := 412.85712, [8,13].EmptyDist := 1410.0, [8,13].FullDist := 1276.2882, [8,13].Carbon_mLperL := 20.108566, [8,13].Slurry_Weight := -10.52187, [8,13].Sample_Tank := 8, [8,13].Carbon_Height := 133.71179, [8,13].Sample_FlowRate := 2.2523706, [8,13].Sample_FillTime := 7.800001, [8,13].DisplacedCarbonVol := 3623.3555, [8,13].DisplacedCarbonMass := 1811.6777, [8,13].SampleDuration := 1025, [8,14].Run_ID := 2646, [8,14].Carbon_VOL_ml := 275.36453, [8,14].Carbon_MASS := 137.68227, [8,14].Carbon_DIST := 7.9062386, [8,14].Hour := 10, [8,14].Min := 57, [8,14].Day := 20, [8,14].Month := 11, [8,14].Year := 2021, [8,14].Sample_DO := 4.959754, [8,14].Sample_pH := 9.204817, [8,14].Sample_VOL := 17.414383, [8,14].Density := 410.59213, [8,14].EmptyDist := 1410.0, [8,14].FullDist := 1305.7773, [8,14].Carbon_mLperL := 15.812477, [8,14].Slurry_Weight := -10.52187, [8,14].Sample_Tank := 8, [8,14].Carbon_Height := 104.22266, [8,14].Sample_FlowRate := 2.1926947, [8,14].Sample_FillTime := 7.942001, [8,14].DisplacedCarbonVol := 2773.7546, [8,14].DisplacedCarbonMass := 1386.8773, [8,14].SampleDuration := 1024, [8,15].Run_ID := 2636, [8,15].Carbon_VOL_ml := 294.3845, [8,15].Carbon_MASS := 147.19225, [8,15].Carbon_DIST := 8.540514, [8,15].Hour := 8, [8,15].Min := 23, [8,15].Day := 20, [8,15].Month := 11, [8,15].Year := 2021, [8,15].Sample_DO := 4.9527187, [8,15].Sample_pH := 9.247381, [8,15].Sample_VOL := 17.234589, [8,15].Density := 407.94955,
        [8,15].EmptyDist := 1410.0, [8,15].FullDist := 1298.5785, [8,15].Carbon_mLperL := 17.081028, [8,15].Slurry_Weight := -10.52187, [8,15].Sample_Tank := 8, [8,15].Carbon_Height := 111.42151, [8,15].Sample_FlowRate := 2.2979448, [8,15].Sample_FillTime := 7.500001, [8,15].DisplacedCarbonVol := 3140.1008, [8,15].DisplacedCarbonMass := 1570.0504, [8,15].SampleDuration := 1033, [8,16].Run_ID := 2626, [8,16].Carbon_VOL_ml := 316.57123, [8,16].Carbon_MASS := 158.28561, [8,16].Carbon_DIST := 9.490637, [8,16].Hour := 5, [8,16].Min := 21, [8,16].Day := 20, [8,16].Month := 11, [8,16].Year := 2021, [8,16].Sample_DO := 4.818126, [8,16].Sample_pH := 9.262283, [8,16].Sample_VOL := 16.678082, [8,16].Density := 399.77032, [8,16].EmptyDist := 1410.0, [8,16].FullDist := 1290.181, [8,16].Carbon_mLperL := 18.981274, [8,16].Slurry_Weight := -10.52187, [8,16].Sample_Tank := 8, [8,16].Carbon_Height := 119.81897, [8,16].Sample_FlowRate := 2.3630035, [8,16].Sample_FillTime := 7.058001, [8,16].DisplacedCarbonVol := 3588.2253, [8,16].DisplacedCarbonMass := 1794.1127, [8,16].SampleDuration := 1025, [8,17].Run_ID := 2617, [8,17].Carbon_VOL_ml := 326.02493, [8,17].Carbon_MASS := 163.01247, [8,17].Carbon_DIST := 8.985302, [8,17].Hour := 3, [8,17].Min := 7, [8,17].Day := 20, [8,17].Month := 11, [8,17].Year := 2021, [8,17].Sample_DO := 5.0574718, [8,17].Sample_pH := 9.290899, [8,17].Sample_VOL := 18.142124, [8,17].Density := 421.28806, [8,17].EmptyDist := 1410.0, [8,17].FullDist := 1286.6029, [8,17].Carbon_mLperL := 17.970604, [8,17].Slurry_Weight := -10.52187, [8,17].Sample_Tank := 8, [8,17].Carbon_Height := 123.397095, [8,17].Sample_FlowRate := 2.4189496, [8,17].Sample_FillTime := 7.500001, [8,17].DisplacedCarbonVol := 3477.5989, [8,17].DisplacedCarbonMass := 1738.7994, [8,17].SampleDuration := 1025, [8,18].Run_ID := 2607,
        [8,18].Carbon_VOL_ml := 329.29175, [8,18].Carbon_MASS := 164.64587, [8,18].Carbon_DIST := 9.964061, [8,18].Min := 31, [8,18].Day := 20, [8,18].Month := 11, [8,18].Year := 2021, [8,18].Sample_DO := 4.5051317, [8,18].Sample_pH := 9.316484, [8,18].Sample_VOL := 16.523973, [8,18].Density := 397.50534, [8,18].EmptyDist := 1410.0, [8,18].FullDist := 1285.3665, [8,18].Carbon_mLperL := 19.928122, [8,18].Slurry_Weight := -10.52187, [8,18].Sample_Tank := 8, [8,18].Carbon_Height := 124.633545, [8,18].Sample_FlowRate := 2.3947785, [8,18].Sample_FillTime := 6.900001, [8,18].DisplacedCarbonVol := 3817.8748, [8,18].DisplacedCarbonMass := 1908.9374, [8,18].SampleDuration := 1024, [8,19].Run_ID := 2599, [8,19].Carbon_VOL_ml := 316.19617, [8,19].Carbon_MASS := 158.09808, [8,19].Carbon_DIST := 8.814251, [8,19].Hour := 22, [8,19].Min := 34, [8,19].Day := 19, [8,19].Month := 11, [8,19].Year := 2021, [8,19].Sample_DO := 3.9676359, [8,19].Sample_pH := 9.33816, [8,19].Sample_VOL := 17.936644, [8,19].Density := 418.268, [8,19].EmptyDist := 1410.0, [8,19].FullDist := 1290.323, [8,19].Carbon_mLperL := 17.628502, [8,19].Slurry_Weight := -10.52187, [8,19].Sample_Tank := 8, [8,19].Carbon_Height := 119.677, [8,19].Sample_FlowRate := 2.599513, [8,19].Sample_FillTime := 6.900001, [8,19].DisplacedCarbonVol := 3666.0417, [8,19].DisplacedCarbonMass := 1833.0209, [8,19].SampleDuration := 1024);   // Sample Result Historical
   CS_Rules : DINT[17] := ([0] := 1, [1] := 1, [2] := 1, [3] := 1, [4] := 1, [5] := 1, [6] := 1, [7] := 1, [16] := 1);
   CS_SampleSeq : DINT[129] := ([0] := 1, [1] := 2, [2] := 3, [3] := 4, [4] := 5, [5] := 6, [6] := 7, [7] := 8);
   CS_Seq : GEK_Sequence := (Mode.Cfg_PCmdClear := 1, Mode.Cfg_OvrdOverLock := 1, Mode.Cfg_ProgDefault := 1, Mode.Val := 8, Mode.Sts_Prog := 1, Mode.Sts_ProgOperSel := 1, Mode.Rdy_MAcq := 1, Mode.Rdy_OAcq := 1, POC.In_Cfg_BatchContinous := 1, POC.Sts_Stopped := 1, POC.In_Stopped := 1, POC.In_StepNum := 13, POC.Out_NewStepNum := 13, POC.Sts_Skipped := 1, POC.In_MaxStepNum := 23, POC.In_Intlk2OK := 1, SeqTimer[0].PRE := 2147483647, Group_ProgAcq_Req := 1);
   CS_Seq_ControlStop : BOOL;
   CS_Seq_CrashStop : BOOL;
   CS_SeqCheckSum1 : DINT := 11111111;
   CS_SeqCheckSum2 : DINT;
   CS_STRINGParams : STRING_20[10] := ([0] := 'CS007', [2] := 'MK6', [3] := '192.168.50.200', [4] := '192.168.50.201', [5] := '192.168.50.205', [6] := '192.168.50.206', [7] := '192.168.50.253', [8] := '-', [9] := 'test');
        [6]   // Transmitter IP
        [5]   // Valve IP
        [7]   // eWON IP
        [0]   // Project Code
        [3]   // PLC IP
        [4]   // HMI IP
        [2]   // Serial Number
        [1]   // Site Name
        [8]   // PC IP
   CS_Tank : CS_TankParams[20] := ([0].Sample_Cnt := 4, [0].Online := 1, [0].From := -9, [0].To := -9, [0].PurgeLow := 1, [1].Run_ID := 2784, [1].Sample_Cnt := 1067, [1].Sample_Time := 200, [1].NoFill_TimeOut := 200, [1].Purge_Time := 200, [1].Online := 1, [1].Name := 'Tank1', [1].CarbonSP := 100.0, [1].To := 2, [1].Volume := 237.0, [1].LiquidDensity := 1.0, [1].SolidsDensity := 2.83, [1].PurgeVolume := 1000.0, [2].Run_ID := 2762, [2].Sample_Cnt := 930, [2].Sample_Time := 200, [2].NoFill_TimeOut := 200, [2].Purge_Time := 200, [2].Name := 'Tank2', [2].CarbonSP := 2.6, [2].From := 1, [2].To := 2, [2].PumpRunTime := 2.6, [2].Volume := 233.0, [2].TotalCarbonMass := 1210.1985, [2].LiquidDensity := 1.0, [2].SolidsDensity := 2.83, [2].PurgeVolume := 1000.0, [3].Run_ID := 2786, [3].Sample_Cnt := 919, [3].Sample_Time := 250, [3].NoFill_TimeOut := 200, [3].Purge_Time := 200, [3].Online := 1, [3].Name := 'Tank3', [3].CarbonSP := 100.0, [3].From := 2, [3].To := 4, [3].Volume := 229.0, [3].LiquidDensity := 1.0, [3].SolidsDensity := 2.83, [3].PurgeVolume := 1000.0, [4].Run_ID := 2788, [4].Sample_Cnt := 827, [4].Sample_Time := 250, [4].NoFill_TimeOut := 150, [4].Purge_Time := 200, [4].Online := 1, [4].Name := 'Tank4', [4].CarbonSP := 100.0, [4].From := 3, [4].To := 5, [4].Volume := 226.0, [4].LiquidDensity := 1.0, [4].SolidsDensity := 2.83,
        [4].PurgeVolume := 1000.0, [5].Run_ID := 2790, [5].Sample_Cnt := 1454, [5].Sample_Time := 250, [5].NoFill_TimeOut := 200, [5].Purge_Time := 90, [5].Online := 1, [5].Name := 'Tank5', [5].CarbonSP := 100.0, [5].From := 4, [5].To := 6, [5].Volume := 129.0, [5].TotalCarbonMass := 232.69676, [5].LiquidDensity := 1.0, [5].SolidsDensity := 2.83, [5].PurgeVolume := 1000.0, [6].Run_ID := 2791, [6].Sample_Cnt := 936, [6].Sample_Time := 250, [6].NoFill_TimeOut := 200, [6].Purge_Time := 90, [6].Online := 1, [6].Name := 'Tank6', [6].CarbonSP := 100.0, [6].From := 5, [6].To := 7, [6].Volume := 135.0, [6].LiquidDensity := 1.0, [6].SolidsDensity := 2.83, [6].PurgeVolume := 1000.0, [7].Run_ID := 2780, [7].Sample_Cnt := 911, [7].Sample_Time := 250, [7].NoFill_TimeOut := 200, [7].Purge_Time := 250, [7].Online := 1, [7].Name := 'Tank7', [7].CarbonSP := 100.0, [7].From := 6, [7].To := 8, [7].Volume := 134.0, [7].LiquidDensity := 1.0, [7].SolidsDensity := 2.83, [7].PurgeVolume := 1000.0, [8].Run_ID := 2782, [8].Sample_Cnt := 879, [8].Sample_Time := 200, [8].NoFill_TimeOut := 200, [8].Purge_Time := 250, [8].Online := 1, [8].Name := 'Tank8', [8].CarbonSP := 100.0, [8].From := 7, [8].To := 9, [8].Volume := 133.0, [8].LiquidDensity := 1.0, [8].SolidsDensity := 2.83, [8].PurgeVolume := 1000.0, [9].Run_ID := 6449, [9].Sample_Cnt := 578,
        [9].Sample_Time := 40, [9].NoFill_TimeOut := 60, [9].Purge_Time := 60, [9].Name := 'Tank9', [9].CarbonSP := 100.0, [9].From := 8, [9].To := 10, [9].Volume := 131.0, [9].TotalCarbonMass := 1302.9784, [9].LiquidDensity := 1.0, [9].SolidsDensity := 2.83, [9].PurgeVolume := 1000.0, [10].Run_ID := 6450, [10].Sample_Cnt := 624, [10].Sample_Time := 35, [10].NoFill_TimeOut := 60, [10].Purge_Time := 60, [10].Name := 'Tank10', [10].CarbonSP := 100.0, [10].From := 9, [10].To := 11, [10].Volume := 137.0, [10].TotalCarbonMass := 1045.5265, [10].LiquidDensity := 1.0, [10].SolidsDensity := 2.83, [10].PurgeVolume := 1000.0, [11].Run_ID := 1724, [11].Sample_Cnt := 110, [11].Sample_Time := 5, [11].NoFill_TimeOut := 60, [11].Purge_Time := 60, [11].Name := 'TNK11', [11].LiquidDensity := 1.0, [11].SolidsDensity := 2.83, [11].LeachOnly := 1, [11].PurgeVolume := 10.0, [12].Run_ID := 1725, [12].Sample_Cnt := 110, [12].Sample_Time := 5, [12].NoFill_TimeOut := 60, [12].Purge_Time := 60, [12].Name := 'TNK12', [12].LiquidDensity := 1.0, [12].SolidsDensity := 2.83, [12].PurgeVolume := 10.0, [13].Run_ID := 1726, [13].Sample_Cnt := 109, [13].Sample_Time := 5, [13].NoFill_TimeOut := 60, [13].Purge_Time := 60, [13].Name := 'TNK13', [13].LiquidDensity := 1.0, [13].SolidsDensity := 2.83, [13].LeachOnly := 1, [13].PurgeVolume := 10.0, [14].Run_ID := 1652, [14].Sample_Cnt := 106, [14].Sample_Time := 5, [14].NoFill_TimeOut := 60, [14].Purge_Time := 60,
        [14].Name := 'TNK14', [14].LiquidDensity := 1.0, [14].SolidsDensity := 2.83, [14].PurgeVolume := 10.0, [15].Run_ID := 1653, [15].Sample_Cnt := 103, [15].Sample_Time := 5, [15].NoFill_TimeOut := 60, [15].Purge_Time := 60, [15].Name := 'TNK15', [15].LiquidDensity := 1.0, [15].SolidsDensity := 2.83, [15].LeachOnly := 1, [15].PurgeVolume := 10.0, [16].Run_ID := 1654, [16].Sample_Cnt := 104, [16].Sample_Time := 5, [16].NoFill_TimeOut := 60, [16].Purge_Time := 60, [16].Name := 'TNK16', [16].LiquidDensity := 1.0, [16].SolidsDensity := 2.83, [16].PurgeVolume := 10.0);
   CS_TankOrder : DINT[17] := ([0] := 1, [1] := 2, [2] := 3, [3] := 4, [4] := 5, [5] := 6, [6] := 7, [7] := 8, [8] := 9, [9] := 10, [10] := 11, [11] := 12, [12] := 13, [13] := 14, [14] := 15, [15] := 16, [16] := 16);
   CS_Timer : TIMER[80] := ([0].PRE := 1000, [0].ACC := 1042, [0].EN := 1, [0].DN := 1, [2].PRE := 200000, [3].PRE := 5000, [4].PRE := 2000, [5].PRE := 10000, [6].PRE := 5000, [7].PRE := 200000, [8].PRE := 200000, [9].PRE := 150000, [10].PRE := 200000, [11].PRE := 200000, [12].PRE := 200000, [13].PRE := 200000, [14].PRE := 60000, [15].PRE := 60000, [16].PRE := 60000, [17].PRE := 90000, [18].PRE := 30000, [19].PRE := 45000, [20].PRE := 45000, [21].PRE := 60000, [22].PRE := 5000, [23].PRE := 20000, [24].PRE := 5000, [25].PRE := 3000, [26].PRE := 3000, [39].PRE := 4000, [40].PRE := 2000, [41].PRE := 20000, [42].PRE := 10000, [42].ACC := 10057, [42].EN := 1, [42].DN := 1, [43].PRE := 3000, [44].PRE := 2147483647, [45].PRE := 5000, [46].PRE := 10000, [46].ACC := 10043, [46].EN := 1, [46].DN := 1, [47].PRE := 10000, [48].PRE := 5000, [49].PRE := 10000, [49].ACC := 10057, [49].EN := 1, [49].DN := 1, [50].PRE := 4000, [51].PRE := 60000, [52].PRE := 60000, [53].PRE := 60000, [54].PRE := 60000, [55].PRE := 60000, [56].PRE := 60000, [57].PRE := 30000, [58].PRE := 5000, [59].PRE := 60000, [60].PRE := 180000,
        [61].PRE := 5000, [62].PRE := 9999999, [62].ACC := 8273857, [62].EN := 1, [62].TT := 1, [63].PRE := 180000, [63].ACC := 180000, [63].EN := 1, [63].DN := 1, [64].PRE := 2000, [64].ACC := 2100, [64].EN := 1, [64].DN := 1, [65].PRE := 1000, [66].PRE := 30000, [67].PRE := 3000, [68].PRE := 3000, [69].PRE := 10000, [70].PRE := 120000, [71].PRE := 3000, [72].PRE := 120000, [73].PRE := 2000, [74].PRE := 10000, [76].PRE := 30000, [77].PRE := 600000, [77].ACC := 157, [77].EN := 1, [77].DN := 1);
        [50]   // Top wash delay timer
        [55]   // Step 6 - Solution Fill Time Out Alarm Timer Tank 15
        [56]   // Step 6 - Solution Fill Time Out Alarm Timer Tank 16
        [10]   // Step 6 - Solution Fill Time Out Alarm Timer Tank 5
        [0]   // DB Timer for Start button
        [20]   // Manual Smaple Wash Time
        [6]   // Step 1 - Step 1 DB timer
        [70]   // Step 13 Laser Watchdog
        [16]   // Step 1 Hopper Levels Are not OK Alarm
        [25]   // Delete backup log Timer
        [17]   // Purge Water Timer (XV11)
        [26]   // DataLog2 Debounce Timer
        [78]   // AutoStart Timer
        [3]   // Low Air Pressure DB Timer
        [18]   // Bottom Wash Timer (XV15)
        [28]   // Transfer Pump 1 Run on Time
        [29]   // Transfer Pump 2 Run on Time
        [30]   // Transfer Pump 3 Run on Time
        [31]   // Transfer Pump 4 Run on Time
        [32]   // Transfer Pump 5 Run on Time
        [33]   // Transfer Pump 6 Run on Time
        [34]   // Transfer Pump 7 Run on Time
        [35]   // Transfer Pump 8 Run on Time
        [36]   // Transfer Pump 9 Run on Time
        [66]   // XRF auto sequence watch dog
        [72]   // Step 1 Laser Flap watch dog
        [43]   // XRF Start Debounce Timer
        [45]   // XV-12 Inlet Purge Timer
        [60]   // XRF Power up delay timer
        [79]   // Spare
        [11]   // Step 6 - Solution Fill Time Out Alarm Timer Tank 6
        [49]   // XRF HeartbeatPC timer
        [27]   // Transfer Feed Pump Run on Time
        [68]   // Sample overfill alarm debounce
        [4]   // Purge Water Flow DB Timer
        [46]   // IDLE Leak Check Timer
        [21]   // Manual Sample Purge Timer
        [47]   // Water Leak Detection Timer
        [62]   // XRF Power up record timer
        [71]   // carbon and result push db
        [12]   // Step 6 - Solution Fill Time Out Alarm Timer Tank 7
        [13]   // Step 6 - Solution Fill Time Out Alarm Timer Tank 8
        [2]   // Step 6 - Solution Fill Time Out Alarm Timer Tank 1
        [1]   // Step 1 - Periodic Sampling Time
        [74]   // Discharge S1
        [75]   // Discharge S2
        [76]   // Discharge S3
        [40]   // Air shot timer
        [22]   // Manual Sample Valve Open Time
        [38]   // Transfer Pump Discharge Run on Time
        [48]   // XRF Power Button Hold Time
        [5]   // Step 6 - Level Check Stablising Timer
        [14]   // Step 6 -Solution Fill Time Out Alarm Timer Tank 9
        [7]   // Step 6- Solution Fill Time Out Alarm Timer Tank 2
        [15]   // Step 6 - Solution Fill Time Out Alarm Timer Tank 10
        [8]   // Step 6 - Solution Fill Time Out Alarm Timer Tank 3
        [9]   // Step 6 - Solution Fill Time Out Alarm Timer Tank 4
        [61]   // XRF Power up button delay timer
        [65]   // XRF auto sequence start delay
        [58]   // XRF Batch Test Water Timer
        [39]   // Bottom wash valve delay time 4 seconds.
        [63]   // XRF expected power up time
        [51]   // Step 6 - Solution Fill Time Out Alarm Timer Tank 11
        [24]   // Data Log Debounce
        [41]   // XV21-30 cycle timer
        [67]   // Laser PVbad debounce
        [44]   // Sample Fill Timer
        [53]   // Step 6 - Solution Fill Time Out Alarm Timer Tank 13
        [42]   // XRF Heartbeat timer
        [57]   // Pegged Screen Timer
        [59]   // XRF Batch Test Delay to XRF test Timer
        [69]   // Alarm Debounce Laser Compartment dirty
        [64]   // XRF Running debounce timer
        [23]   // Delete Log Timer
        [73]   // Tank Change Debounce Timer
        [19]   // Manual Sample Discharge Time
        [37]   // Transfer Pump 10 Run on Time
        [52]   // Step 6 - Solution Fill Time Out Alarm Timer Tank 12
        [54]   // Step 6 - Solution Fill Time Out Alarm Timer Tank 14
        [77]   // XRF software WatchDog 10 minuts then move on and triger reboot
   CS_Timer2 : TIMER[20] := ([0].PRE := 600000);
   CS_XRF : XRF := (Run_ID := 2791, Sts_CommLoss := 1, Mode := 1, Sts_Powered := 1, Modes.Cfg_PCmdClear := 1, Modes.Cfg_OvrdOverLock := 1, Modes.Sts_Oper := 1);
        .ModbusINT_OUT[0]   // Beam 1 Min
        .ModbusINT_OUT[1]   // Beam 1 Max
        .ModbusBOOL_OUT[1]   // Stop Test 0x0003
        .ModbusINT_OUT[2]   // Beam 2 Min
        .ModbusINT_OUT[3]   // Beam 2 Max
        .Results[11]   // Hg Error
        .Results[13]   // Pb Error
        .Results[15]   // Zn Error
        .Results[17]   // Sn Error
        .Results[0]   // Au ppm
        .ModbusBOOL_IN[1]   // Sts Ready 0x00002
        .Results[2]   // As ppm
        .ModbusBOOL_IN[2]   // Heartbeat 0x00003
        .Results[4]   // Cu ppm
        .Results[6]   // Fe ppm
        .Results[8]   // Ag ppm
        .ModbusBOOL_OUT[0]   // Start Test 0x0002
        .Results[19]   // Ca Error
        .Results[21]   // Mg Error
        .ModbusBOOL_IN[0]   // HeartbeatPC 0x00001
        .Results[23]   // Al Error
        .Results[26]   // P ppm
        .Results[28]   // S ppm
        .Results[25]   // Si Error
        .ModbusBOOL_OUT[2]   // Set Beam Configuration 0x0004
        .Results[10]   // Hg ppm
        .Results[27]   // P error
        .Results[29]   // S Error
        .Results[31]   // K Error
        .Results[35]   // V Error
        .Results[33]   // Ti Error
        .Results[37]   // Cr Error
        .Results[12]   // Pb ppm
        .Results[30]   // K ppm
        .Results[34]   // V ppm
        .ModbusBOOL_IN   // Modbus Feedback BOOL
        .Results[39]   // Mn Error
        .Results[41]   // Co Error
        .ModbusINT_OUT   // Modbus INT Commands
        .Results[43]   // Ni Error
        .ModbusDINT_IN[0]   // Package Id
        .Results[14]   // Zn ppm
        .Results[16]   // Sn ppm
        .Results[18]   // Ca ppm
        .Results[1]   // Au Error
        .Results[20]   // Mg ppm
        .Results[22]   // Al ppm
        .Results[24]   // Si ppm
        .Results[32]   // Ti ppm
        .Results[36]   // Cr ppm
        .Results[38]   // Mn ppm
        .Results[3]   // As Error
        .Results[40]   // Co ppm
        .Results[42]   // Ni ppm
        .Results[5]   // Cu Error
        .Results[7]   // Fe Error
        .Results[9]   // Ag Error
        .ModbusBOOL_OUT   // Modbus Command BOOL
        .ModbusDINT_IN   // Modbus INT Feedbacks
        .ModbusDINT_IN[1]   // Stop Reason ID
   CS_XRF_DetTemp : REAL := -29.999039;   // Used in ewon for data records
   CS_XRF_Elements : LinearModelXRF := (Au_Scaled := 1253.0, Au_ErrScaled := 21.0, Au_Raw := 3842.0, Au_ErrRaw := 36.0, Au_Model[0].A := 2.45814, Au_Model[1].A := 0.13172387, Au_Model[1].B := 9.2587185, Mg_ErrScaled := 36423.0, Mg_ErrRaw := 36423.0, Mg_Model[0].A := 1.0, Mg_Model[1].A := 1.0, Al_Scaled := 1457.0, Al_ErrScaled := 202.0, Al_Raw := 1457.0, Al_ErrRaw := 202.0, Al_Model[0].A := 1.0, Al_Model[1].A := 1.0, Si_Scaled := 647.0, Si_ErrScaled := 68.0, Si_Raw := 647.0, Si_ErrRaw := 68.0, Si_Model[0].A := 1.0, Si_Model[1].A := 1.0, S_Scaled := 204.0, S_ErrScaled := 27.0, S_Raw := 204.0, S_ErrRaw := 27.0, S_Model[0].A := 1.0, S_Model[1].A := 1.0, K_ErrScaled := 2737.0, K_ErrRaw := 2737.0, K_Model[0].A := 1.0, K_Model[1].A := 1.0, Ca_Scaled := 4029.0, Ca_ErrScaled := 28.0, Ca_Raw := 4029.0, Ca_ErrRaw := 28.0, Ca_Model[0].A := 1.0, Ca_Model[1].A := 1.0, Ti_Scaled := 158.0, Ti_ErrScaled := 52.0, Ti_Raw := 158.0, Ti_ErrRaw := 52.0, Ti_Model[0].A := 1.0, Ti_Model[1].A := 1.0, V_ErrScaled := 22.0, V_ErrRaw := 22.0, V_Model[0].A := 1.0, V_Model[1].A := 1.0, Cr_ErrScaled := 12.0, Cr_ErrRaw := 12.0, Cr_Model[0].A := 1.0, Cr_Model[1].A := 1.0, Mn_Scaled := 57.0, Mn_ErrScaled := 6.0, Mn_Raw := 57.0, Mn_ErrRaw := 6.0, Mn_Model[0].A := 1.0, Mn_Model[1].A := 1.0, Fe_Scaled := 4280.0,
        Fe_ErrScaled := 30.0, Fe_Raw := 4280.0, Fe_ErrRaw := 30.0, Fe_Model[0].A := 1.0, Fe_Model[1].A := 1.0, Co_ErrScaled := 13.0, Co_ErrRaw := 13.0, Co_Model[0].A := 1.0, Co_Model[1].A := 1.0, Ni_Scaled := 121.0, Ni_ErrScaled := 3.0, Ni_Raw := 121.0, Ni_ErrRaw := 3.0, Ni_Model[0].A := 1.0, Ni_Model[1].A := 1.0, Cu_Scaled := 192.0, Cu_ErrScaled := 4.0, Cu_Raw := 192.0, Cu_ErrRaw := 4.0, Cu_Model[0].A := 1.0, Cu_Model[1].A := 1.0, Zn_ErrScaled := 5.0, Zn_ErrRaw := 5.0, Zn_Model[0].A := 1.0, Zn_Model[1].A := 1.0, As_ErrScaled := 1.0, As_ErrRaw := 1.0, As_Model[0].A := 1.0, As_Model[1].A := 1.0, Se_Scaled := 19.0, Se_ErrScaled := 1.0, Se_Raw := 19.0, Se_ErrRaw := 1.0, Se_Model[0].A := 1.0, Se_Model[1].A := 1.0, Rb_ErrScaled := 1.0, Rb_ErrRaw := 1.0, Rb_Model[0].A := 1.0, Rb_Model[1].A := 1.0, Sr_Scaled := 41.0, Sr_Raw := 41.0, Sr_Model[0].A := 1.0, Sr_Model[1].A := 1.0, Y_Scaled := 4.0, Y_Raw := 4.0, Y_Model[0].A := 1.0, Y_Model[1].A := 1.0, Zr_Scaled := 1.0, Zr_ErrScaled := 1.0, Zr_Raw := 1.0, Zr_ErrRaw := 1.0, Zr_Model[0].A := 1.0, Zr_Model[1].A := 1.0, Nb_ErrScaled := 1.0, Nb_ErrRaw := 1.0, Nb_Model[0].A := 1.0, Nb_Model[1].A := 1.0, Mo_ErrScaled := 2.0, Mo_ErrRaw := 2.0, Mo_Model[0].A := 1.0,
        Mo_Model[1].A := 1.0, Ag_Scaled := 12.0, Ag_ErrScaled := 1.0, Ag_Raw := 12.0, Ag_ErrRaw := 1.0, Ag_Model[0].A := 1.0, Ag_Model[1].A := 1.0, Cd_ErrScaled := 8.0, Cd_ErrRaw := 8.0, Cd_Model[0].A := 1.0, Cd_Model[1].A := 1.0, Sn_ErrScaled := 10.0, Sn_ErrRaw := 10.0, Sn_Model[0].A := 1.0, Sn_Model[1].A := 1.0, Sb_ErrScaled := 15.0, Sb_ErrRaw := 15.0, Sb_Model[0].A := 1.0, Sb_Model[1].A := 1.0, Ba_Model[0].A := 1.0, Ba_Model[1].A := 1.0, La_Model[0].A := 1.0, La_Model[1].A := 1.0, Ce_Model[0].A := 1.0, Ce_Model[1].A := 1.0, Pr_Model[0].A := 1.0, Pr_Model[1].A := 1.0, Nd_Model[0].A := 1.0, Nd_Model[1].A := 1.0, W_ErrScaled := 43.0, W_ErrRaw := 43.0, W_Model[0].A := 1.0, W_Model[1].A := 1.0, Hg_ErrScaled := 14.0, Hg_ErrRaw := 14.0, Hg_Model[0].A := 1.0, Hg_Model[1].A := 1.0, Pb_Scaled := 7.0, Pb_ErrScaled := 1.0, Pb_Raw := 7.0, Pb_ErrRaw := 1.0, Pb_Model[0].A := 1.0, Pb_Model[1].A := 1.0, Bi_ErrScaled := 21.0, Bi_ErrRaw := 21.0, Bi_Model[0].A := 1.0, Bi_Model[1].A := 1.0, Th_Scaled := 27.0, Th_ErrScaled := 2.0, Th_Raw := 27.0, Th_ErrRaw := 2.0, Th_Model[0].A := 1.0, Th_Model[1].A := 1.0, U_Scaled := 5.0, U_ErrScaled := 1.0, U_Raw := 5.0, U_ErrRaw := 1.0, U_Model[0].A := 1.0, U_Model[1].A := 1.0, LE_Model[0].A := 1.0,
        LE_Model[1].A := 1.0);   // Linear model 0 is inital factory model and 1 is trimming model
   CS_XRF_Elements_Saved : LinearModelXRF := (Au_ErrRaw := 3.0, Au_Model[0].A := 2.458138, Au_Model[1].A := 0.6388, Mg_ErrRaw := 45425.0, Mg_Model[0].A := 1.0, Mg_Model[1].A := 1.0, Al_Raw := 10650.0, Al_ErrRaw := 818.0, Al_Model[0].A := 1.0, Al_Model[1].A := 1.0, Si_Raw := 12131.0, Si_ErrRaw := 361.0, Si_Model[0].A := 1.0, Si_Model[1].A := 1.0, S_Raw := 8117.0, S_ErrRaw := 137.0, S_Model[0].A := 1.0, S_Model[1].A := 1.0, K_ErrRaw := 3655.0, K_Model[0].A := 1.0, K_Model[1].A := 1.0, Ca_Raw := 2670.0, Ca_ErrRaw := 73.0, Ca_Model[0].A := 1.0, Ca_Model[1].A := 1.0, Ti_ErrRaw := 3962.0, Ti_Model[0].A := 1.0, Ti_Model[1].A := 1.0, V_ErrRaw := 41.0, V_Model[0].A := 1.0, V_Model[1].A := 1.0, Cr_Raw := 1106.0, Cr_ErrRaw := 46.0, Cr_Model[0].A := 1.0, Cr_Model[1].A := 1.0, Mn_Raw := 221.0, Mn_ErrRaw := 22.0, Mn_Model[0].A := 1.0, Mn_Model[1].A := 1.0, Fe_Raw := 4115.0, Fe_ErrRaw := 57.0, Fe_Model[0].A := 1.0, Fe_Model[1].A := 1.0, Co_Raw := 99.0, Co_ErrRaw := 15.0, Co_Model[0].A := 1.0, Co_Model[1].A := 1.0, Ni_Raw := 227.0, Ni_ErrRaw := 9.0, Ni_Model[0].A := 1.0, Ni_Model[1].A := 1.0, Cu_Raw := 33.0, Cu_ErrRaw := 4.0, Cu_Model[0].A := 1.0, Cu_Model[1].A := 1.0, Zn_ErrRaw := 4.0, Zn_Model[0].A := 1.0, Zn_Model[1].A := 1.0, As_ErrRaw := 2.0, As_Model[0].A := 1.0,
